(* CODESYS project stdnov.library
   Company: National Oilwell Varco
   DefaultNamespace: stdNOV
   Version: 1.0.0.2936
   Placeholder: stdNOV
   Author: AACD
   Title: stdNOV

Project tree, tasks and I/O mapping:
  libraries: SysTimeCore, * (System); Tc2_EtherCAT, * (Beckhoff Automation GmbH); Tc2_ModbusSrv, * (Beckhoff Automation GmbH); Tc2_Standard, * (Beckhoff Automation GmbH); Tc2_System, * (Beckhoff Automation GmbH); Tc2_Utilities, 3.3.41.0 (Beckhoff Automation GmbH); Util, * (System)
  10 Documentation/
  20 Program Organization Units/
    Alarms/
      function f_AlarmCode [ST]
      function f_DeviceId [ST]
      function f_FaultCode [ST]
      function f_GetFaultCodePriority [ST]
      function block fb_AlarmHandler [ST]: Clear, FB_exit, FB_init, GetAlarmCodeIndex, GetAlarms, GetNumOfActiveAlarms, GetNumOfAlarms, GetNumOfDeviceId, GetNumRegisteredCodes, GetRegisteredAlarmCodeDWORDListPointer, GetRegisteredAlarmCodeListPointer, GetRegisteredDeviceComponentIdListPointer, GetRegisteredDeviceElementIdListPointer, GetRegisteredFaultCondiitionIdListPointer, GetRegisteredFaultPriorityIdListPointer, Init, RegisterAlarmCode, Set
      function block fb_AlarmInterface [ST]: FB_exit, FB_init, ResetAlarms, UpdateAlarms
      function block fb_AlarmMonitor [ST]: CheckLimits, DisableLimit, EnableLimit, FB_exit, FB_init, GetState, InitAlarm, Monitor, MonitorBool, MonitorInt, MonitorReal, SetDelayOn, SetLimitBool, SetLimitInt, SetLimitReal
    Command Interface/
      Interfaces/
        interface i_commandHandler: CommandDone, CommandRunning, CommandStart, Fault, Reset
      function block fb_CommandInterface [ST]: CMD_ClearCommandBuffer, CMD_Fault, CMD_Init, CMD_IsCommandValid, CMD_Reset, CMD_SendCommand, CMD_SetTraceTable, CMD_TRACE, CMD_UpdateCommandInterface, ExecuteAction
    Control Functions/
      PID Functions/
        function block PID_StandAlone [ST]: Execute, FB_init, GetGains, GetLimits, init, Reset, SetGains, SetLimits
        function block PID_StandAlone_AntiWindup [ST]: Execute, FB_init, GetConfig, init, Reset, SetConfig
        function block PID_StandAlone_Stuck [ST]: Execute, FB_init, GetGains, GetLimits, init, Reset, SetGains, SetLimits
    Equipment Functions/
      TriStateValve/
        ENUMS/
          data type TriStateValveFsmAction
          data type TriStateValveFsmEvent
          data type TriStateValveFsmState
        function block fb_AnalogFeedbackValve [ST]: CloseValve, FB_exit, FB_init, InitAlarms, IsClosed, IsOpened, IsShifting, IsShiftingError, OpenValve
        function block fb_DigitalFeedbackDualActionValve [ST]: CloseValve, FB_exit, FB_init, InitAlarms, IsClosed, IsOpened, IsShifting, IsShiftingError, OpenValve
        function block fb_DigitalFeedbackSingleActionValve [ST]: CloseValve, FB_exit, FB_init, InitAlarms, IsClosed, IsOpened, IsShifting, IsShiftingError, OpenValve
        function block fb_DigitalFeedbackValve [ST]: CloseValve, FB_exit, FB_init, InitAlarms, IsClosed, IsOpened, IsShifting, IsShiftingError, OpenValve
        function block fb_NoFeedbackValve [ST]: CloseValve, FB_exit, FB_init, IsClosed, IsOpened, IsShifting, IsShiftingError, OpenValve
        function block fb_TriStateValve [ST]: CloseValve, ExecuteAction, FB_exit, FB_init, OpenValve
    FSM/
      Interfaces/
        interface i_actionHandler: ExecuteAction
      function block fb_FSM [ST]: FB_exit, FB_init, FSM_ASSERT, FSM_GetCurrentAction, FSM_GetCurrentEvent, FSM_GetCurrentState, FSM_GetNextState, FSM_GetPreviousState, FSM_ProcessEvent, FSM_ProcessEventWithParms, FSM_Reset, FSM_SetAlwaysChangeState, FSM_SetConditionalState, FSM_SetDebugTraceTable, FSM_SetErrorState, FSM_TRACE
    Input-Output Functions/
      function block fb_AnalogOutputActuator [ST]: AbortCal, Arm, Disarm, Fault, FB_exit, FB_init, GetDevId, GetMaxInput, GetMaxOutput, GetMinInput, GetMinOutput, GetZeroCalValue, InitAlarms, IsZeroCalRunning, ZeroCal
      function block fb_AnalogTransducer [ST]: AbortCal, Arm, Disarm, Fault, FB_exit, FB_init, GetDevId, GetMaxOutput, GetMinOutput, GetWireBreakStatus, GetZeroCalValue, InitAlarms, IsZeroCalRunning, ZeroCal
      function block fb_FreqTransducer [ST]: FaultHandlerSetOrClear, FB_init, GetDevId, InitAlarms
    Instrument-Controller Functions/
      function block fb_Densitometer [ST]: CalculateUserkFact, GetCorrectedDensitySGU, GetDensityRange_MinMax, GetRawDensity, GetUserKFact, InitAlarms, SetDensityRange_MinMax, SetRawDensity, setUserKFact
      function block fb_ENDP_Analog [ST]: FB_init, Get_UserAlarms, GetConfigData, GetRange_MinMax, InitAlarms, Scale, Set_Hysteresis, SetRange_MinMax, SetRange_UserAlarms
      function block fb_ENDP_AnalogCalPressure [ST]: CalculateUserKFactor, CalibrateHighDataPoint, CalibrateLowDataPoint, ClearCalibration, FB_Exit, FB_Init, GetConfigData, GetCorrectedPressure, GetLowerCalDataPoint, GetPressureRange, GetRawPressure, GetUpperCalDataPoint, GetUserAlarms, GetUserKFactor, InitAlarms, SetHysteresis, SetLowerCalDataPoint, SetPressureRange, SetRangeUserAlarms, SetRawPressure, SetUpperCalDataPoint, SetUserKFactor
      function block fb_ENDP_AnalogDensitometer [ST]: FB_exit, FB_init
      function block fb_ENDP_AnalogFlowmeter [ST]: CalibrateHighDataPoint, CalibrateLowDataPoint, ClearCalibration, FB_exit, FB_init, GetLowerCalDataPoint, GetUpperCalDataPoint, SetLowerCalDataPoint, SetUpperCalDataPoint
      function block fb_ENDP_Freq_Tachometer [ST]: FB_init
      function block fb_ENDP_FreqFlowmeter [ST]: FB_exit, FB_init, GetKFact, GetPPR, GetTimebase, SetKFact, SetPPR, SetTimebase
      function block fb_ENDP_SimulatedDensitometer [ST]: FB_exit, FB_init, SetSimDensity
      function block fb_ENDP_SimulatedFlowMeter [ST]: FB_exit, FB_init, SetSimFlow
      function block fb_FlowMeter [ST]: CalculateUserKFact, GetCorrectedFlow, GetFlowRange_MinMax, GetRawFlow, GetUserAlarms, GetUserKFact, GetVolumeTotal1, GetVolumeTotal2, GetVolumeTotal3, InitAlarms, PauseVolumeTotal1, PauseVolumeTotal2, PauseVolumeTotal3, ResetVolumeTotal1, ResetVolumeTotal2, ResetVolumeTotal3, ResumeVolumeTotal1, ResumeVolumeTotal2, ResumeVolumeTotal3, SetFlowRange_MinMax, SetRawFlow, SetUserAlarms, SetUserKFact
      function block fb_Indicator [ST]: FB_exit, FB_init, Off, On
      function block fb_STARTP_ControlActuator [ST]: FB_init, GetConfigData, GetRange_MinMax, Scale, Set_Hysteresis, SetRange_MinMax
      function block fb_Switch [ST]: Equals, FB_exit, FB_init, GetDebounce, SetDebounce
    Interlock Functions/
      function block fb_NOVInterlock [ST]: FB_exit, FB_init, InitAlarms
    Modbus/
      function block fb_ModbusError [FBD]
      function block fb_ModbusServer [FBD]: afterAccess, beforeAccess, FB_exit, FB_init, GetCoilPointer, GetDiscreteInputPointer, GetHoldingRegisterPointer, GetInputRegisterPointer, IsClientConnected, UpdateConnectionList
      function block fb_ReadHoldingRegisters [FBD]
      function block fb_ReadInputRegisters [FBD]
      function block fb_WriteHoldingRegisters [FBD]
    Process Calculation Functions/
      function f_CalculateDensityPPAfromSGU [ST]
      function f_CalculateDensityPPGfromSGU [ST]
    Testing Functions/
      function block FB_CNTRLSYS_RESPONSE [ST]
      function block fb_TriStateValveSimulator [ST]
    Utility Functions/
      Conversion Functions/
        function F_SPLIT_REGISTERS [ST]
        function F_STATUS_WORD_TO_WORD [ST]
      Statistic Functions/
        function block FB_RUNNING_AVG [ST]
      function f_LinearScale [ST]
      function block fb_Clock [ST]
      function block fb_ElapsedTime [ST]: FB_exit, FB_init, GetElapsedLTime, GetElapsedTime, StartNow
      function block fb_ElapseTimer [ST]: FB_exit, FB_init, Freeze, Initialize, Reset
      function block fb_FilterExp [ST]: FB_exit, FB_init, GetSampleSize, Initialize, SetSampleSize
      function block fb_GetCycleTime [ST]
      function block fb_TriggerTimer [ST]
      function block Logger [ST]: getCount, LogPoint
      function block Totalizer [ST]: Disable, Enable, FB_Init, Reset, SetTotal
  40 Data Types/
    Alarm Interface Types/
      data type TAlarm
      data type TAlarmData
    Alarm Types/
      global variables GLOBAL_ALARMS
      data type TAlarmCode
      data type TAlarmLimit
      data type TAlarmMessage
      data type TAlarmMonitorType
      data type TAlarmType
      data type TComponentId
      data type TDeviceId
      data type TElementId
      data type TFaultCode
      data type TFaultCondition
      data type TFaultPriority
      data type UAlarmCode
      data type UDeviceId
      data type UFaultCode
    Command Interface/
      data type Command_FsmAction
      data type Command_FsmDebugTableEntry
      data type Command_FsmEvent
      data type Command_FsmState
      data type TControlCommand
      data type TControlCommandBuffer
      data type TControlCommandParms
      data type TControlCommandResponse
      data type TControlResponse
      data type TControlResponseMessage
    Equipment Types/
      data type TValveShutoff
      data type TValveTriStatePosition
    FSM Types/
      global variables GLOBAL_FSM
      data type TFsmAction
      data type TFsmDebugTableEntry
      data type TFsmError
      data type TFsmEvent
      data type TFsmEventDesc
      data type TFsmEventQIndex
      data type TFsmState
    Generic Types/
      data type ST_Bits
    Input-Output Types/
      data type AI_ChannelInputs
      data type AO_ChannelOutputs
      data type Freq_ChannelInput
    Instrument-Controller Types/
      global variables GLOBAL_INSTRUMENTS
      data type HmiGaugeState
      data type TCalibrationDataPoint
      data type TEndPoint
      data type TEndPointConfig
      data type TEnuHmiGaugeState
    Interlock Types/
      data type THMINOVInterlock
      data type TNOVInterlockCmdBypassInWORD
      data type TNOVInterlockIn
      data type TNOVInterlockStatusInWORD
      data type TNOVInterlockStatusOut
      data type TNOVInterlockStatusOutWORD
    Modbus Types/
      global variables GLOBAL_MODBUS
      data type TModbusServerConfig
      data type TModbusServerConnection
      data type TModbusTargetConfig
    Utility Types/
      data type DataPoint
      data type TGenericStatusWord
    global variables GLOBAL_CONSTANTS
  80 Status/
  Project Information/
    function F_GetCompany [ST]
    function F_GetTitle [ST]
    function F_GetVersion [ST]
  Version/
    global variables Global_Version
*)

// 20 Program Organization Units/Equipment Functions/TriStateValve/ENUMS/TriStateValveFsmAction
{attribute 'qualified_only'}
//{attribute 'strict'}
TYPE TriStateValveFsmAction :
(
	FsmAction_None := FSM_ACTION_NONE,		(*0*)
	FsmAction_ValveEnabled := 1,			(*1*)
	FsmAction_ValveDisabled,				(*2*)
	FsmAction_ValveOpen,					(*3*)
	FsmAction_ValveClose,					(*4*)
	FsmAction_ValveOpened,					(*5*)
	FsmAction_ValveClosed,					(*6*)
	FsmAction_ValveShiftTimerExpired,		(*7*)
	FsmAction_ValvePositionMismatch,		(*8*)
	NUM_FsmTriStateValveActions				(*9*)
) BYTE;
END_TYPE

// 20 Program Organization Units/Equipment Functions/TriStateValve/ENUMS/TriStateValveFsmEvent
{attribute 'qualified_only'}
//{attribute 'strict'}
TYPE TriStateValveFsmEvent :
(
	FsmEvent_ValveEnable := 0,			(*0*)
	FsmEvent_ValveDisable,				(*1*)
	FsmEvent_ValveOpen,					(*2*)
	FsmEvent_ValveClose,				(*3*)
	FsmEvent_ValveOpened,				(*4*)
	FsmEvent_ValveClosed,				(*5*)
	FsmEvent_ValveShiftTimerExpired,	(*6*)
	FsmEvent_ValvePositionMismatch,		(*7*)
	NUM_FsmTriStateValveEvents			(*8*)
) BYTE;
END_TYPE

// 20 Program Organization Units/Equipment Functions/TriStateValve/ENUMS/TriStateValveFsmState
{attribute 'qualified_only'}
//{attribute 'strict'}
TYPE TriStateValveFsmState :
(
	FsmState_Error := 0,			(*0*)
	FsmState_ValveOff,				(*1*)
	FsmState_ValveClosed,			(*2*)
	FsmState_ValveOpened,  			(*3*)
	FsmState_ValveShifting,			(*4*)
	NUM_FsmTriStateValveStates		(*5*)
) BYTE;
END_TYPE

// 40 Data Types/Alarm Interface Types/TAlarm
TYPE TAlarm :
STRUCT
	code	: UDINT;
	state	: BOOL;
	ack		: BOOL;
	message	: STRING(95);
END_STRUCT
END_TYPE

// 40 Data Types/Alarm Interface Types/TAlarmData
TYPE TAlarmData :
STRUCT
	NumOfAlarms			: INT;
	NumOfActiveAlarms	: INT;
	RefreshAlarms		: BOOL;
	AlarmState			: INT;
	Alarm				: ARRAY[0.._ALARM_ARRAY_MAX_SIZE] OF TAlarm;
END_STRUCT
END_TYPE

// 40 Data Types/Alarm Types/TAlarmCode
// I have made the DeviceId the MSB so that when sorting the alarm list
// all similar deviceId's will be grouped together. <JAISON>
TYPE TAlarmCode :
STRUCT
	faultCode	: UFaultCode;	// LSB (16 bits)
	devId		: UDeviceId;	// MSB (16 bits)
END_STRUCT
END_TYPE

// 40 Data Types/Alarm Types/TAlarmLimit
TYPE TAlarmLimit :
STRUCT
	limitOn		: LREAL;
	limitOff	: LREAL;
	enable		: BOOL;
	monitorType	: TAlarmMonitorType;
END_STRUCT
END_TYPE

// 40 Data Types/Alarm Types/TAlarmMessage
TYPE TAlarmMessage :
STRUCT
	code	: UAlarmCode;			// 32 bits
	msg		: STRING;
END_STRUCT
END_TYPE

// 40 Data Types/Alarm Types/TAlarmMonitorType
{attribute 'qualified_only'}
{attribute 'strict'}
TYPE TAlarmMonitorType :
(
	lower_limit := 0,
	upper_limit
);
END_TYPE

// 40 Data Types/Alarm Types/TAlarmType
TYPE TAlarmType :
STRUCT
	code	: UAlarmCode;
	state	: BOOL;
	message	: STRING;
END_STRUCT
END_TYPE

// 40 Data Types/Alarm Types/TComponentId
TYPE TComponentId : BYTE; END_TYPE

// 40 Data Types/Alarm Types/TDeviceId
// Device Ids (16 bits)
TYPE TDeviceId :
STRUCT
	element		: BYTE;	// LSB (8 bits)
	component	: BYTE;	// MSB (8 bits)
END_STRUCT
END_TYPE

// 40 Data Types/Alarm Types/TElementId
TYPE TElementId : BYTE; END_TYPE

// 40 Data Types/Alarm Types/TFaultCode
// Fault Codes (16 bits)
TYPE TFaultCode :
STRUCT
	condition	: BYTE; // LSB (8 bits)
	priority	: BYTE; // MSB (8 bits) 	
END_STRUCT
END_TYPE

// 40 Data Types/Alarm Types/TFaultCondition
{attribute 'qualified_only'}
//{attribute 'strict'}
TYPE TFaultCondition :
(
	SelfTest := 0,
	Generic,
	Check,
	Config,
	UnderLimit,
	OverLimit,
	Protect,
	UnderWarning,
	OverWarning,
	TimeOut,
	HwError,
	ShortCircuit,
	UnderRange,
	OverRange,
	Shutdown,
	Stop,
	Interlock
) BYTE;
END_TYPE

// 40 Data Types/Alarm Types/TFaultPriority
{attribute 'qualified_only'}
//{attribute 'strict'}
TYPE TFaultPriority :
(
	// The 2 most significant bits of the fault code are reserved for severity
	// This has now been explanded to 8 bits however the Hex values are kept for
	// backwards compatibility AND to give space for future priority additions. <JAISON>
	Information := 16#00,	// 0
	Warning		:= 16#40,	// 64
	Error		:= 16#80,	// 128
	Reserved	:= 16#C0,	// 192
	Critical	:= 16#FF	// 255
) BYTE;
END_TYPE

// 40 Data Types/Alarm Types/UAlarmCode
TYPE UAlarmCode :
UNION
	code		: TAlarmCode;
	code_UDINT	: UDINT;
	code_DWORD	: DWORD;
	code_BYTES	: ARRAY[1..4] OF BYTE;   
    code_BITS	: ARRAY[1..4] OF ST_Bits;
END_UNION
END_TYPE

// 40 Data Types/Alarm Types/UDeviceId
TYPE UDeviceId :
UNION
	devId		: TDeviceId;
	devId_UINT	: UINT;
	devId_WORD	: WORD;
	devId_BYTES	: ARRAY[1..2] OF BYTE;  
    devId_BITS	: ARRAY[1..2] OF ST_Bits;
END_UNION
END_TYPE

// 40 Data Types/Alarm Types/UFaultCode
TYPE UFaultCode :
UNION
	faultcode		: TFaultCode;
	faultcode_UINT	: UINT;
	faultcode_WORD	: WORD;
	faultcode_BYTES	: ARRAY[1..2] OF BYTE;   
    faultcode_BITS	: ARRAY[1..2] OF ST_Bits;
END_UNION
END_TYPE

// 40 Data Types/Command Interface/Command_FsmAction
{attribute 'qualified_only'}
//{attribute 'strict'}
TYPE Command_FsmAction :
(
	FsmAction_None := FSM_ACTION_NONE,				(*0*)
	FsmAction_EnableControl := 1,					(*1*)
	FsmAction_DisableControl,						(*2*)
	FsmAction_RunCommand,							(*3*)
	FsmAction_CommandDone,							(*4*)
	FsmAction_Fault,								(*5*)
	FsmAction_Reset,								(*6*)
	NUM_FsmCommandInterfaceActions					(*7*)
) BYTE;
END_TYPE

// 40 Data Types/Command Interface/Command_FsmDebugTableEntry
TYPE Command_FsmDebugTableEntry :
STRUCT
	state		: Command_FsmState;	// State transitioning to
	event		: Command_FsmEvent;	// Event causing the transition
	timeInState	: UDINT;			// Elapsed time since the last event (ms)
END_STRUCT
END_TYPE

// 40 Data Types/Command Interface/Command_FsmEvent
{attribute 'qualified_only'}
//{attribute 'strict'}
TYPE Command_FsmEvent :
(
	FsmEvent_ControlEnable := 0,		(*0*)
	FsmEvent_ControlDisable,			(*1*)
	FsmEvent_RunCommand,				(*2*)
	FsmEvent_CommandDone,				(*3*)
	FsmEvent_Fault,						(*4*)
	FsmEvent_Reset,						(*5*)
	NUM_FsmCommandInterfaceEvents		(*6*)
) BYTE;
END_TYPE

// 40 Data Types/Command Interface/Command_FsmState
{attribute 'qualified_only'}
//{attribute 'strict'}
TYPE Command_FsmState :
(
	FsmState_ControlFault := 0,			(*0*)
	FsmState_ControlDisabled,			(*1*)
	FsmState_CommandRunning,			(*2*)
	FsmState_ControlReady,				(*3*)
	NUM_FsmCommandInterfaceStates		(*4*)	
) BYTE;
END_TYPE

// 40 Data Types/Command Interface/TControlCommand
{attribute 'strict'}
TYPE TControlCommand : INT; END_TYPE

// 40 Data Types/Command Interface/TControlCommandBuffer
TYPE TControlCommandBuffer :
STRUCT
	command		: TControlCommand;
	parms		: TControlCommandParms;
	response	: TControlCommandResponse;
END_STRUCT
END_TYPE

// 40 Data Types/Command Interface/TControlCommandParms
TYPE TControlCommandParms : ARRAY[1..12] OF WORD; END_TYPE

// 40 Data Types/Command Interface/TControlCommandResponse
TYPE TControlCommandResponse :
STRUCT
	response	: TControlResponse;
	message		: TControlResponseMessage;
END_STRUCT
END_TYPE

// 40 Data Types/Command Interface/TControlResponse
{attribute 'strict'}
TYPE TControlResponse : INT; END_TYPE

// 40 Data Types/Command Interface/TControlResponseMessage
TYPE TControlResponseMessage : STRING(27); END_TYPE

// 40 Data Types/Equipment Types/TValveShutoff
TYPE TValveShutoff :
STRUCT
	Open	: BOOL;
	Close	: BOOL;
END_STRUCT
END_TYPE

// 40 Data Types/Equipment Types/TValveTriStatePosition
{attribute 'qualified_only'}
{attribute 'strict'}
TYPE TValveTriStatePosition :
(
	PosClosed := 0,
	PosOpened,
	PosUnknown
);
END_TYPE

// 40 Data Types/FSM Types/TFsmAction
TYPE TFsmAction : BYTE; END_TYPE

// 40 Data Types/FSM Types/TFsmDebugTableEntry
TYPE TFsmDebugTableEntry :
STRUCT
	state		: TFsmState;	// State transitioning to
	event		: TFsmEvent;	// Event causing the transition
	timeInState	: UDINT;		// Elapsed time since the last event (ms)
END_STRUCT
END_TYPE

// 40 Data Types/FSM Types/TFsmError
{attribute 'qualified_only'}
TYPE TFsmError :
(
	FSM_ERROR_NONE := 0,
	FSM_INVALID_NEXT_STATE,
	FSM_PARM_SIZE_ERROR,
	FSM_EVENT_Q_SIZE_ERROR,
	FSM_INVALID_EVENT_ERROR,
	FSM_INVALID_ACTION,
	FSM_INVALID_CONDITIONAL_STATE,
	FSM_INVALID_ERROR_STATE
) BYTE;
END_TYPE

// 40 Data Types/FSM Types/TFsmEvent
{attribute 'strict'}
TYPE TFsmEvent : BYTE; END_TYPE

// 40 Data Types/FSM Types/TFsmEventDesc
TYPE TFsmEventDesc :
STRUCT
	event		: BYTE;
	parms		: POINTER TO BYTE;
	parmSize	: UINT;
END_STRUCT
END_TYPE

// 40 Data Types/FSM Types/TFsmEventQIndex
TYPE TFsmEventQIndex : UINT; END_TYPE

// 40 Data Types/FSM Types/TFsmState
TYPE TFsmState : BYTE; END_TYPE

// 40 Data Types/Generic Types/ST_Bits
TYPE ST_Bits :
STRUCT
	bBit1  : BIT;
    bBit2  : BIT;
    bBit3  : BIT;
    bBit4  : BIT;
    bBit5  : BIT;
    bBit6  : BIT;
    bBit7  : BIT;
    bBit8  : BIT;   
END_STRUCT
END_TYPE

// 40 Data Types/Input-Output Types/AI_ChannelInputs
TYPE AI_ChannelInputs :
STRUCT
	value				: INT;
	underRange			: BOOL;
	overRange			: BOOL;
	error				: BOOL;
	shortCircuit		: BOOL;
END_STRUCT
END_TYPE

// 40 Data Types/Input-Output Types/AO_ChannelOutputs
TYPE AO_ChannelOutputs :
STRUCT
	value				: INT;
END_STRUCT
END_TYPE

// 40 Data Types/Input-Output Types/Freq_ChannelInput
TYPE Freq_ChannelInput :
STRUCT
	value		: DINT;
	//error		: BOOL;
END_STRUCT
END_TYPE

// 40 Data Types/Instrument-Controller Types/HmiGaugeState
{attribute 'qualified_only'}
{attribute 'strict'}
TYPE HmiGaugeState :
(
	LowAlarm := -2,
	LowWarning := -1,
	No_Alarm := 0,
	HighWarning := 1,
	HighAlarm := 2
);
END_TYPE

// 40 Data Types/Instrument-Controller Types/TCalibrationDataPoint
TYPE TCalibrationDataPoint :
STRUCT
	yValue	: REAL;
	xValue	: REAL;
END_STRUCT
END_TYPE

// 40 Data Types/Instrument-Controller Types/TEndPoint
TYPE TEndPoint :
STRUCT
	Value	:	REAL;
	State	:	INT;
END_STRUCT
END_TYPE

// 40 Data Types/Instrument-Controller Types/TEndPointConfig
TYPE TEndPointConfig :
STRUCT
	MinValue	:	REAL;
	MaxValue	:	REAL;
	OffsetValue	:	REAL;
	LowLimit	:	REAL;
	HighLimit	:	REAL;
	LowWarning	:	REAL;
	HighWarning	:	REAL;
END_STRUCT
END_TYPE

// 40 Data Types/Instrument-Controller Types/TEnuHmiGaugeState
{attribute 'qualified_only'}
{attribute 'strict'}
TYPE TEnuHmiGaugeState :
(
	LowAlarm 	:= -2,
	LowWarning 	:= -1,
	No_Alarm 	:= 0,
	HighWarning	:= 1,
	HighAlarm 	:= 2
);
END_TYPE

// 40 Data Types/Interlock Types/THMINOVInterlock
/// WORD ALLIGNED (2 WORDS) <GRAHAM>
TYPE THMINOVInterlock :
STRUCT
	
	//HMIInterlockBypass : TNOVInterlockCmdBypassInWORD;	// INTLK DynIn, for future use, HMI may have the ability to override in the future
	HMIInterlockProcessed: TNOVInterlockStatusOutWORD; 		// INTLK DynOut
	
END_STRUCT
END_TYPE

// 40 Data Types/Interlock Types/TNOVInterlockCmdBypassInWORD
/// this input commmand data structure word is for future use (not used currently) <GRAHAM>
TYPE TNOVInterlockCmdBypassInWORD :
STRUCT
	
	IntlkBypassALL	: BIT; // Bypass/override all interlocks command input
	Intlk01Bypass	: BIT; // TRUE = (OVERRIDE ACTIVE), FALSE = (OVERRIDE NOT ACTIVE)
	Intlk02Bypass	: BIT; // TRUE = (OVERRIDE ACTIVE), FALSE = (OVERRIDE NOT ACTIVE)
	Intlk03Bypass	: BIT; // TRUE = (OVERRIDE ACTIVE), FALSE = (OVERRIDE NOT ACTIVE)
	Intlk04Bypass	: BIT; // TRUE = (OVERRIDE ACTIVE), FALSE = (OVERRIDE NOT ACTIVE)
	Intlk05Bypass	: BIT; // TRUE = (OVERRIDE ACTIVE), FALSE = (OVERRIDE NOT ACTIVE)
	Intlk06Bypass	: BIT; // TRUE = (OVERRIDE ACTIVE), FALSE = (OVERRIDE NOT ACTIVE)
	Intlk07Bypass	: BIT; // TRUE = (OVERRIDE ACTIVE), FALSE = (OVERRIDE NOT ACTIVE)
	Intlk08Bypass	: BIT; // TRUE = (OVERRIDE ACTIVE), FALSE = (OVERRIDE NOT ACTIVE)
	Intlk09Bypass	: BIT; // TRUE = (OVERRIDE ACTIVE), FALSE = (OVERRIDE NOT ACTIVE)
	Intlk10Bypass	: BIT; // TRUE = (OVERRIDE ACTIVE), FALSE = (OVERRIDE NOT ACTIVE)
	Intlk11Bypass	: BIT; // TRUE = (OVERRIDE ACTIVE), FALSE = (OVERRIDE NOT ACTIVE)
	Intlk12Bypass	: BIT; // TRUE = (OVERRIDE ACTIVE), FALSE = (OVERRIDE NOT ACTIVE)
	Intlk13Bypass	: BIT; // TRUE = (OVERRIDE ACTIVE), FALSE = (OVERRIDE NOT ACTIVE)
	IntlkBypassNONE	: BIT; // Do not Bypass/override any interlocks command input
	Bit15			: BIT; // Spare Bit command input
END_STRUCT
END_TYPE

// 40 Data Types/Interlock Types/TNOVInterlockIn
/// WORD ALLIGNED (2 WORDS), this input data structure is for future use (not used currently) <GRAHAM>
TYPE TNOVInterlockIn :
STRUCT
	
	InterlockStatus		: TNOVInterlockStatusInWORD;	// INTLK In (from NOV or NSA interlocks)
	//InterlockBypass	: TNOVInterlockCmdBypassInWORD;	// INTLK In (from an external device), for future use
	
END_STRUCT
END_TYPE

// 40 Data Types/Interlock Types/TNOVInterlockStatusInWORD
/// this input structure data word is for future use (not used currently) <GRAHAM>
TYPE TNOVInterlockStatusInWORD :
STRUCT
	
	Bit0	: BIT; // Not Defined
	Intlk01	: BIT; // TRUE = (INTLK SATISFIED), FALSE = (INTLK NOT SATISFIED)
	Intlk02	: BIT; // TRUE = (INTLK SATISFIED), FALSE = (INTLK NOT SATISFIED)
	Intlk03	: BIT; // TRUE = (INTLK SATISFIED), FALSE = (INTLK NOT SATISFIED)
	Intlk04	: BIT; // TRUE = (INTLK SATISFIED), FALSE = (INTLK NOT SATISFIED) 
	Intlk05	: BIT; // TRUE = (INTLK SATISFIED), FALSE = (INTLK NOT SATISFIED)
	Intlk06	: BIT; // TRUE = (INTLK SATISFIED), FALSE = (INTLK NOT SATISFIED)
	Intlk07	: BIT; // TRUE = (INTLK SATISFIED), FALSE = (INTLK NOT SATISFIED)
	Intlk08	: BIT; // TRUE = (INTLK SATISFIED), FALSE = (INTLK NOT SATISFIED)
	Intlk09	: BIT; // TRUE = (INTLK SATISFIED), FALSE = (INTLK NOT SATISFIED)
	Intlk10	: BIT; // TRUE = (INTLK SATISFIED), FALSE = (INTLK NOT SATISFIED)
	Intlk11	: BIT; // TRUE = (INTLK SATISFIED), FALSE = (INTLK NOT SATISFIED)
	Intlk12	: BIT; // TRUE = (INTLK SATISFIED), FALSE = (INTLK NOT SATISFIED)
	Intlk13	: BIT; // TRUE = (INTLK SATISFIED), FALSE = (INTLK NOT SATISFIED)
	Bit14	: BIT; // Not defined
	Bit15	: BIT; // Not defined
	
END_STRUCT
END_TYPE

// 40 Data Types/Interlock Types/TNOVInterlockStatusOut
/// WORD ALLIGNED (1 WORD), // this seperate output structure data word is for future use (not used currently) <GRAHAM>
TYPE TNOVInterlockStatusOut :
STRUCT
	
	InterlockProcessed: TNOVInterlockStatusOutWORD; // INTLK DynOut
END_STRUCT
END_TYPE

// 40 Data Types/Interlock Types/TNOVInterlockStatusOutWORD
TYPE TNOVInterlockStatusOutWORD :
STRUCT
	IntlkOK_NoBypass	: BIT; 	// All interlocks are Ok with no bypasses/overrides
	Intlk01				: BIT; // TRUE = (INTLK IS TRUE OR OVERRIDE IS TRUE IF OVERRIDE IS ACTIVE, FALSE = (INTLK IS FALSE AND OVERRIDE IS FALSE IF OVERRIDE IS ACTIVE)
	Intlk02				: BIT; // TRUE = (INTLK IS TRUE OR OVERRIDE IS TRUE IF OVERRIDE IS ACTIVE, FALSE = (INTLK IS FALSE AND OVERRIDE IS FALSE IF OVERRIDE IS ACTIVE)
	Intlk03				: BIT; // TRUE = (INTLK IS TRUE OR OVERRIDE IS TRUE IF OVERRIDE IS ACTIVE, FALSE = (INTLK IS FALSE AND OVERRIDE IS FALSE IF OVERRIDE IS ACTIVE)
	Intlk04				: BIT; // TRUE = (INTLK IS TRUE OR OVERRIDE IS TRUE IF OVERRIDE IS ACTIVE, FALSE = (INTLK IS FALSE AND OVERRIDE IS FALSE IF OVERRIDE IS ACTIVE)
	Intlk05				: BIT; // TRUE = (INTLK IS TRUE OR OVERRIDE IS TRUE IF OVERRIDE IS ACTIVE, FALSE = (INTLK IS FALSE AND OVERRIDE IS FALSE IF OVERRIDE IS ACTIVE)
	Intlk06				: BIT; // TRUE = (INTLK IS TRUE OR OVERRIDE IS TRUE IF OVERRIDE IS ACTIVE, FALSE = (INTLK IS FALSE AND OVERRIDE IS FALSE IF OVERRIDE IS ACTIVE)
	Intlk07				: BIT; // TRUE = (INTLK IS TRUE OR OVERRIDE IS TRUE IF OVERRIDE IS ACTIVE, FALSE = (INTLK IS FALSE AND OVERRIDE IS FALSE IF OVERRIDE IS ACTIVE)
	Intlk08				: BIT; // TRUE = (INTLK IS TRUE OR OVERRIDE IS TRUE IF OVERRIDE IS ACTIVE, FALSE = (INTLK IS FALSE AND OVERRIDE IS FALSE IF OVERRIDE IS ACTIVE)
	Intlk09				: BIT; // TRUE = (INTLK IS TRUE OR OVERRIDE IS TRUE IF OVERRIDE IS ACTIVE, FALSE = (INTLK IS FALSE AND OVERRIDE IS FALSE IF OVERRIDE IS ACTIVE)
	Intlk10				: BIT; // TRUE = (INTLK IS TRUE OR OVERRIDE IS TRUE IF OVERRIDE IS ACTIVE, FALSE = (INTLK IS FALSE AND OVERRIDE IS FALSE IF OVERRIDE IS ACTIVE)
	Intlk11				: BIT; // TRUE = (INTLK IS TRUE OR OVERRIDE IS TRUE IF OVERRIDE IS ACTIVE, FALSE = (INTLK IS FALSE AND OVERRIDE IS FALSE IF OVERRIDE IS ACTIVE)
	Intlk12				: BIT; // TRUE = (INTLK IS TRUE OR OVERRIDE IS TRUE IF OVERRIDE IS ACTIVE, FALSE = (INTLK IS FALSE AND OVERRIDE IS FALSE IF OVERRIDE IS ACTIVE)
	Intlk13				: BIT; // TRUE = (INTLK IS TRUE OR OVERRIDE IS TRUE IF OVERRIDE IS ACTIVE, FALSE = (INTLK IS FALSE AND OVERRIDE IS FALSE IF OVERRIDE IS ACTIVE)
	IntlkOK_WithBypass	: BIT; // All interlocks are Ok with bypasses/overrides
	Bit15				: BIT; // Not defined
END_STRUCT
END_TYPE

// 40 Data Types/Modbus Types/TModbusServerConfig
TYPE TModbusServerConfig :
STRUCT
	xInstalled				: BOOL;
	tTimeOut				: TIME;
END_STRUCT
END_TYPE

// 40 Data Types/Modbus Types/TModbusServerConnection
TYPE TModbusServerConnection :
STRUCT
	xActive					: BOOL;
	ipAddress				: STRING(20);
	bUnitId					: BYTE;		
	bFunctionCode			: BYTE;
	wReadAddress			: WORD;
	uiReadQuantity			: UINT;
	uiReadQuantityTotal		: UINT;
	wWriteAddress			: WORD;
	uiWriteQuantity			: UINT;
	uiWriteQuantityTotal	: UINT;
	commLossTimer			: TON;
END_STRUCT
END_TYPE

// 40 Data Types/Modbus Types/TModbusTargetConfig
TYPE TModbusTargetConfig :
STRUCT
	xInstalled				: BOOL;			// Not Used
	sIPAddr					: STRING(23);
	wTCPPort				: WORD;
	bUnitID					: BYTE;
	tTimeOut				: TIME;
END_STRUCT
END_TYPE

// 40 Data Types/Utility Types/DataPoint
TYPE DataPoint :
STRUCT
	timestamp: TIME;
	message: STRING(20);
	counter: UINT;
END_STRUCT
END_TYPE

// 40 Data Types/Utility Types/TGenericStatusWord
/// Generic Status Word to handle Word to Bit
TYPE TGenericStatusWord :
STRUCT
	bit0: BIT;
	bit1: BIT;
	bit2: BIT;
	bit3: BIT;
	bit4: BIT;
	bit5: BIT;
	bit6: BIT;
	bit7: BIT;
	bit8: BIT;
	bit9: BIT;
	bit10: BIT;
	bit11: BIT;
	bit12: BIT;
	bit13: BIT;
	bit14: BIT;
	bit15: BIT;
END_STRUCT
END_TYPE

// 40 Data Types/Alarm Types/GLOBAL_ALARMS
{attribute 'global_init_slot' := '49987'}
VAR_GLOBAL CONSTANT
	
	(* --------------------------------------------------------------------------
	Config Parm : _ALARM_ARRAY_MAX_SIZE
	Description : 	This option defines the maximum number of elements defined in 
				 	all of the defined alarm arrays.  This includes the following:
						fb_AlarmHandler/m_alarmList - Internal alarm list
						fb_AlarmInterface/FB_Init/alarmMsg - Static Alarm message array
						fb_AlarmInterface/UpdateAlarms/m_pAlarms - Alarm Interface array
	Notes       : 	This value should be set greater than the maximum number of
					defined alarms in the system.
	-------------------------------------------------------------------------- *)
	_ALARM_ARRAY_MAX_SIZE: UINT := 400;
	
END_VAR

VAR_GLOBAL
	
	// Singleton Alarm handler instantiation
	// Use a pointer to this function block to access its methods
	gAlarmHandler		: fb_AlarmHandler;

END_VAR

// 40 Data Types/FSM Types/GLOBAL_FSM
{attribute 'global_init_slot' := '49987'}
VAR_GLOBAL CONSTANT
	
	(* --------------------------------------------------------------------------
	Config Parm : _FSM_EVENT_Q_SIZE
	Description : This option defines the number of events that can be
   		          stored by the Fsm.
	Notes       : This should be set to the largest queue size for all 
            	  FSMs in the system if optimization is required.
	              Maximum queue size is 256.
	-------------------------------------------------------------------------- *)
	_FSM_EVENT_Q_SIZE: UINT := 32;
	
	(* ---------------------------------------------------------------------------
	Config Parm : _FSM_MAX_PARM_STRUCT_SIZE
	Description : This option defines the maximum number of bytes required
            	  to store event parmeters.      
	Notes       : The size defaults to a large value to allow all event 
            	  parameters to be handled. This should be set to the largest
            	  parameter size for all events for all FSMs in the system if
           	   optimization is required.
	--------------------------------------------------------------------------- *)
	_FSM_MAX_PARM_STRUCT_SIZE: UINT := 512;
	
	(* --------------------------------------------------------------------------
	Config Parm : _FSM_ALLOW_CONDITIONAL_STATES
	Description : This option enables the handling of conditional states.
	Notes       : A conditional state is a state that has state transitions
 	             that can occur from within an action handler.
	-------------------------------------------------------------------------- *)
	_FSM_ALLOW_CONDITIONAL_STATES: BOOL := TRUE;
						
	(* ----------------------------------------------------------------------------
	Const name  : FSM_STATE_CONDITIONAL
	Description : Signifies that the next state is set by an action function 
	Notes       : Used in FSM table definitions
	---------------------------------------------------------------------------- *)
	FSM_STATE_CONDITIONAL: BYTE := 16#7F;

	(* ----------------------------------------------------------------------------
	Const name  : FSM_STATE_INVALID
	Description : Denotes that the state value is invalid
	Notes       : Returned by FSM_GetCurrentState()
	---------------------------------------------------------------------------- *)
	FSM_STATE_INVALID: BYTE := 16#FF;

	(* ----------------------------------------------------------------------------
	Const name  : FSM_EVENT_INVALID
	Description : Signifies that the event is not handled in the state 
	Notes       : Used in FSM table definitions
	---------------------------------------------------------------------------- *)
	FSM_EVENT_INVALID: BYTE := 16#FF;

	(* ----------------------------------------------------------------------------
	Const name  : FSM_ACTION_NONE
	Description : Signifies that no action is required to run
	              in the processing of the current state.
	Notes       : Used in FSM table definitions. For single action tables,
	              informs the FSM to move to the outlined next state.
	---------------------------------------------------------------------------- *)
	FSM_ACTION_NONE: BYTE := 16#00;
	
	(* ----------------------------------------------------------------------------
	Const name  : FSM_ACTION_UNEXPECTED_EVENT
	Description : Signifies that the event is not expected in the state 
	Notes       : Used in FSM table definitions and action handler. 
				  The FSM will not change state when this action is found.
	---------------------------------------------------------------------------- *)
	FSM_ACTION_UNEXPECTED_EVENT: BYTE := 16#FE;
	
	(* ----------------------------------------------------------------------------
	Const name  : FSM_ACTION_ERROR_EVENT
	Description : Signifies that an FSM Assert has failed 
	Notes       : Used in FSM action handler to trap actions required to run
				  on transition to the defined error state.  This will NOT be
				  called if no error state is defined.
	---------------------------------------------------------------------------- *)
	FSM_ACTION_ERROR_EVENT: BYTE := 16#FF;
	
END_VAR

// 40 Data Types/Instrument-Controller Types/GLOBAL_INSTRUMENTS
{attribute 'global_init_slot' := '49987'}
VAR_GLOBAL CONSTANT
	(* --------------------------------------------------------------------------
	Config Parm : NOTUSED
	Description : a flag-type-of-Value passed to ENDPoints to mark that
	              parameter is a Non-Value, rather a flag that is is unused.
				  It is definitely out of range foreseable usable-values,
				  and in addition it has a fraction part to eliminate coincidence.
	Notes       : This removes potential confusion with setting alarmable-limits 
            	  with a barrage of large values like a 100000.0 ...
                  or negatives if parameter is marking a LowAlarm side.
                  Felipe did that as a !quick! solution to place unreachable values
                  and thus mark them as "unused", but later it raised a LOT of questions
                  when we were standardizing that bckhff-code into Codesys as a library
	-------------------------------------------------------------------------- *)
	NOTUSED : REAL := 200001.24681;
	NOTUSED_HIMAX : REAL := (1000000.0);
	NOTUSED_LOMAX : REAL := (-300.0);
	
END_VAR

// 40 Data Types/Modbus Types/GLOBAL_MODBUS
{attribute 'global_init_slot' := '49987'}
VAR_GLOBAL CONSTANT
	
	// Static arrays can have a defined size from 0 - 65535.
	// The array index determines the modbus address for accessing the data. <JAISON>
	// I have left the "Discrete Input" and "Coil" array sizes smaller as its less likely we will use them
	// so no reason to waste memory space. <JAISON>
	DISCRETE_INPUT_ARRAY_SIZE		: UINT := 1;
	COIL_ARRAY_SIZE					: UINT := 1;
	INPUT_REGISTERS_ARRAY_SIZE		: UINT := 65535;
	HOLDING_REGISTERS_ARRAY_SIZE	: UINT := 65535;
	
END_VAR

VAR_GLOBAL
	
	// As long as the PLC Modbus server has been configured with the standard XML these arrays will be mapped to the server.
	// These memory spaces are to be accessed via the pointer using the "Get" routines of the fb_ModbusServer. <JAISON>
	gaxDiscreteInputs				: ARRAY [0..DISCRETE_INPUT_ARRAY_SIZE] OF BOOL;		// Internal modbus server discrete inputs memory space
	gaxCoils						: ARRAY [0..COIL_ARRAY_SIZE] OF BOOL;				// Internal modbus server coils memory space
	gawInputRegisters				: ARRAY [0..INPUT_REGISTERS_ARRAY_SIZE] OF WORD;	// Internal modbus server input register memory space
	gawHoldingRegisters				: ARRAY [0..HOLDING_REGISTERS_ARRAY_SIZE] OF WORD;	// Internal modbus server holding register memory space
	

END_VAR

// 40 Data Types/GLOBAL_CONSTANTS
{attribute 'global_init_slot' := '49987'}
VAR_GLOBAL CONSTANT

	(* --------------------------------------------------------------------------
	Constant	 : _NULL
	Description : This defines a common variable to test for NULL pointers.
	Notes       : 
	-------------------------------------------------------------------------- *)
	_NULL: UINT := 0;
	
	(* C O N V E R S I O N   F A C T O R S *)
	PSI_TO_MPA 						: REAL := 0.00689475729;
	MPA_TO_PSI						: REAL := 145.0377;
	FT3_TO_M3						: REAL := 1/35.3146662127;	//ft^3 to m^3
	M3_TO_FT3						: REAL := 35.3146662127;	//m^3 to ft^3
	SECONDS_IN_MINUTE				: REAL := 60;
	PERCENT_PER_DECIMAL				: REAL := 100;
	GAL_TO_L						: REAL := 3.78541;			//Gallons to Liters
	L_TO_GAL						: REAL := 0.264172;
	MILLI_PER_SECOND				: DINT := 1000;	
	MILLI_PER_MINUTE				: DINT := 60000;
	MILLI_PER_HOUR					: DINT := 3600000;
	LB_TO_DaN						: REAL := 0.444822;
	DaN_TO_LB						: REAL := 2.248089;
	LB_TO_KG						: REAL := 0.453592;
	KG_TO_LB						: REAL := 2.20462;
	FT_TO_M							: REAL := 0.3048;
	M_TO_FT							: REAL := 3.280839895;
	REAL_MAX						: REAL := 3.40282346E+38;
	REAL_MIN						: REAL := 1.179435E-38;
	IN3_TO_GAL						: REAL := 1/231.0;
	SCF_PER_GAL						: REAL := 93.11;			//Standard Cubic Ft (at 1 atm and 70°F) per Gallon of Liquid Nitrogen (LN2)
	PI								: REAL := 3.14159;
	KPA_TO_PSI						: REAL := 0.145038;			

END_VAR

// Version/Global_Version
{attribute 'TcGenerated'}
{attribute 'no-analysis'}
{attribute 'linkalways'}
// This function has been automatically generated from the project information.
VAR_GLOBAL CONSTANT
	{attribute 'const_non_replaced'}
	stLibVersion_stdNOV : ST_LibVersion := (iMajor := 1, iMinor := 0, iBuild := 0, iRevision := 2936, nFlags := 0, sVersion := '1.0.0.2936');
END_VAR

// 20 Program Organization Units/Alarms/f_AlarmCode
(*AUTHOR:			Jaison Schaab*)
(*DATE:				January 21 / 2020*)
(*DESCRIPTION: 		This Function will compose an alarm code from input
					device Id and fault code.*)
(*INPUTS:			devId		-	device Id
					code		-	fault code*)
(*OUTPUTS:			UAlarmCode	-	composed alarm code*)

(*NOTES:			
*)

(*UPDATE: 			March. 22 2021 - Jaison Schaab

					Code Is fully tested and functional.
					
*)

FUNCTION f_AlarmCode : UAlarmCode
VAR_INPUT
	devId	: UDeviceId;
	code	: UFaultCode;
END_VAR
VAR
END_VAR

f_AlarmCode.code.devId.devId 			:= devId.devId;
f_AlarmCode.code.faultCode.faultcode 	:= code.faultcode;

END_FUNCTION

// 20 Program Organization Units/Alarms/f_DeviceId
(*AUTHOR:			Jaison Schaab*)
(*DATE:				January 21 / 2020*)
(*DESCRIPTION: 		This Function will compose a device Id from input
					component Id and element Id.*)
(*INPUTS:			compId		-	component Id
					elemId		-	element Id*)
(*OUTPUTS:			UDeviceId	-	composed device Id*)

(*NOTES:			
*)

(*UPDATE: 			March. 22 2021 - Jaison Schaab

					Code Is fully tested and functional.
					
*)

FUNCTION f_DeviceId : UDeviceId
VAR_INPUT
	compId	: TComponentId;
	elemId	: TElementId;
END_VAR
VAR
END_VAR

f_DeviceId.devId.component 	:= compId;
f_DeviceId.devId.element 	:= elemId;

END_FUNCTION

// 20 Program Organization Units/Alarms/f_FaultCode
(*AUTHOR:			Jaison Schaab*)
(*DATE:				January 21 / 2020*)
(*DESCRIPTION: 		This Function will compose a fault code from input
					fault priority and fault condition.*)
(*INPUTS:			priority	-	fault priority
					condition	-	fault condition*)
					
(*OUTPUTS:			UFaultCode	-	composed fault code*)

(*NOTES:			
*)

(*UPDATE: 			March. 22 2021 - Jaison Schaab

					Code Is fully tested and functional.
					
*)

FUNCTION f_FaultCode : UFaultCode
VAR_INPUT
	priority	: TFaultPriority;
	condition	: TFaultCondition;
END_VAR
VAR
END_VAR

f_FaultCode.faultcode.priority 	:= priority;
f_FaultCode.faultcode.condition := condition;

END_FUNCTION

// 20 Program Organization Units/Alarms/f_GetFaultCodePriority
(*AUTHOR:			Jaison Schaab*)
(*DATE:				January 21 / 2020*)
(*DESCRIPTION: 		This Function will decode and return the priority number 
					for a given fault code input.*)
(*INPUTS:			code	-	fault code*)
(*OUTPUTS:			UINT	-	priority value of the fault code*)

(*NOTES:			This routine was written and intended to be used for
					the purpose of sorting the alarm list by priority.
*)

(*UPDATE: 			March. 22 2021 - Jaison Schaab

					Code Is fully tested and functional.
					
*)

FUNCTION f_GetFaultCodePriority : UINT
VAR_INPUT
	code	: UFaultCode;
END_VAR
VAR
END_VAR

f_GetFaultCodePriority := TO_UINT(SHR((code.faultcode_WORD AND 16#FF00), 8));

END_FUNCTION

// 20 Program Organization Units/Alarms/fb_AlarmHandler
(*AUTHOR:			Jaison Schaab*)
(*DATE:				December 30 / 2019*)
(*DESCRIPTION: 		This Function Block contains the alarm list and all methods
					to interact with it; including Set and Clear.*)
					
(*NOTES:			The alarm list is a static array which contains "_ALARM_ARRAY_MAX_SIZE"
					number of elements, however, not all will be populated.  When the Init
					method is called the alarm list will be initialized with ONLY those alarms
					which have text associated with them.  Use the GetNumOfAlarms method which
					returns the number of configured alarms.  If a SET or CLEAR method is 
					called on a non-existent alarm it will simply be ignored.
*)

(*UPDATE: 			March. 22 2021 - Jaison Schaab

					Code Is fully tested and functional.
					
					A fix had to be made in the "Init" method to pass the alarm message array in as a pointer
					instead of static array.  Beckhoff support is unsure why this was generating a TCOM error,
					however using a pointer fixed the issue and is a more efficient method of passing the array.
					
*)

(*UPDATE: 			March. 18 2021 - Jaison Schaab

					Code Ported from Wago.
					
					Code is NOT YET Operational. There is an issue with sharing memory from within a library
					that is not handled on the beckhoff which could be due to Beckhoff using an older version
					of Codesys from Wago.
*)

(*UPDATE: 			June. 23 2020 - Jaison Schaab

					Added "RegisterAlarmCode" function as well as 6 lists which track all of the
					availible registered alarm codes within the project.  These lists are as 
					follows:
						
						- m_RegAlarmCodeList - List of TAlarmCode
						- m_RegAlarmCodeDWORDList - List of DWORD;
						- m_RegDeviceComponentIdList - List of TComponentId;
						- m_RegDeviceElementIdList - List of TElementId;
						- m_RegFaultPriorityIdList - List of TFaultPriority;
						- m_RegFaultConditionIdList - List of TFaultCondition;
*)

FUNCTION_BLOCK fb_AlarmHandler
VAR_INPUT
END_VAR
VAR_OUTPUT
END_VAR
VAR
	// List of defined alarm codes, states, and messages
	m_alarmList					: ARRAY[0.._ALARM_ARRAY_MAX_SIZE] OF TAlarmType;
	
	m_numAlarms					: UINT;
	m_numActiveAlarms			: UINT;
	
	// Lists of all registered possible alarm codes
	m_RegAlarmCodeList			: ARRAY[1.._ALARM_ARRAY_MAX_SIZE + 1] OF TAlarmCode;
	m_RegAlarmCodeDWORDList		: ARRAY[1.._ALARM_ARRAY_MAX_SIZE + 1] OF DWORD;
	m_RegDeviceComponentIdList	: ARRAY[1.._ALARM_ARRAY_MAX_SIZE + 1] OF TComponentId;
	m_RegDeviceElementIdList	: ARRAY[1.._ALARM_ARRAY_MAX_SIZE + 1] OF TElementId;
	m_RegFaultPriorityIdList	: ARRAY[1.._ALARM_ARRAY_MAX_SIZE + 1] OF TFaultPriority;
	m_RegFaultConditionIdList	: ARRAY[1.._ALARM_ARRAY_MAX_SIZE + 1] OF TFaultCondition;
	
	m_numRegCodes				: UINT;
END_VAR

(* ---------------------------------------------------------------------------
Func name   : 	Clear
Description : 	Clears the state of the input alarm code if it is found
				in the alarm list, also updates the active alarm counter.
Inputs      :	code	- 	alarm code
Returns     : 	None
Notes       : 	
--------------------------------------------------------------------------- *)

METHOD Clear
VAR_INPUT
	code	: UAlarmCode;	// Input alarm code
END_VAR
VAR
	i		: UINT;			// Alarm list index
END_VAR
// Find the specified alarm in the alarm list
i := 0;

WHILE ((i < m_numAlarms) AND (m_alarmList[i].code.code_UDINT <> code.code_UDINT)) DO
	// Incriment to the next alarm message
	i := i + 1;	
END_WHILE

// If the alarm was found and active clear it.
IF ((i < m_numAlarms) AND (m_alarmList[i].state = TRUE)) THEN
	
	// Clear the alarm flag in the alarm list (static map)
	m_alarmList[i].state := FALSE;
	
	// Subtract alarm count from the active alarms
	m_numActiveAlarms := m_numActiveAlarms - 1;

END_IF
END_METHOD

(* ---------------------------------------------------------------------------
Func name   : 	FB_exit
Description : 	Destructor
Inputs      :	None
Returns     : 	None
Notes       : 	
--------------------------------------------------------------------------- *)

METHOD FB_exit
VAR_INPUT
	bInCopyCode : BOOL; // if TRUE, the exit method is called for exiting an instance that is copied afterwards (online change)
END_VAR
// Do nothing
END_METHOD

(* ---------------------------------------------------------------------------
Func name   : 	FB_init
Description : 	Constructor
Inputs      :	None
Returns     : 	None
Notes       : 	
--------------------------------------------------------------------------- *)

METHOD FB_init
VAR_INPUT
	bInitRetains 		: BOOL; // if TRUE, the retain variables are initialized (warm start / cold start)
    bInCopyCode  		: BOOL; // if TRUE, the instance afterwards gets moved into the copy code (online change)
END_VAR
m_numRegCodes := 0;
END_METHOD

(* ---------------------------------------------------------------------------
Func name   : 	GetAlarmCodeIndex
Description : 	Searches the internal alarm list and returns the
				array index of the specified alarm code.
Inputs      :	code	- 	alarm code
Returns     : 	UINT	- 	array index of alarm code
Notes       : 	
--------------------------------------------------------------------------- *)

METHOD GetAlarmCodeIndex : UINT
VAR_INPUT
	code	: UAlarmCode;	// Input alarm code
END_VAR
VAR		
	i		: INT;			// Alarm list index
END_VAR
// Find the specified alarm in the alarm list
i := 0;

// Stop searching once the desired Alarm Code is reached OR the end of the alarm list is found. <JAISON>
WHILE ((i < TO_INT(m_numAlarms)) AND (m_alarmList[i].code.code_UDINT <> code.code_UDINT)) DO
	
	// Incriment to the next alarm message
	i := i + 1;	
END_WHILE

GetAlarmCodeIndex := TO_UINT(i);
END_METHOD

(* ---------------------------------------------------------------------------
Func name   : 	GetAlarms
Description : 	Returns a pointer to the alarm list.
Inputs      :	None
Returns     : 	POINTER TO ARRAY[0.._ALARM_ARRAY_MAX_SIZE] OF AlarmType
Notes       : 	
--------------------------------------------------------------------------- *)

METHOD GetAlarms : POINTER TO ARRAY[0.._ALARM_ARRAY_MAX_SIZE] OF TAlarmType;
VAR_INPUT
END_VAR
GetAlarms := ADR(m_alarmList);
END_METHOD

(* ---------------------------------------------------------------------------
Func name   : 	GetNumOfActiveAlarms
Description : 	Retrieves the number of active alarms in the alarm list.
Inputs      :	None
Returns     : 	UINT	-	the number of active alarms
Notes       : 	
--------------------------------------------------------------------------- *)

METHOD GetNumOfActiveAlarms : UINT
VAR_INPUT
END_VAR
GetNumOfActiveAlarms := m_numActiveAlarms;
END_METHOD

(* ---------------------------------------------------------------------------
Func name   : 	GetNumOfAlarms
Description : 	Retrieves the number of configured alarms in the alarm list.
Inputs      :	None
Returns     : 	UINT	-	the number of alarms in the alarm list
Notes       : 	
--------------------------------------------------------------------------- *)

METHOD GetNumOfAlarms : UINT
VAR_INPUT
END_VAR
GetNumOfAlarms := m_numAlarms;
END_METHOD

(* ---------------------------------------------------------------------------
Func name   : 	GetNumOfDeviceId
Description : 	Searches the internal alarm list and returns the number of
				defined alarms with the input device id.
Inputs      :	devId		- 	input device id
Returns     : 	UINT		- 	the number of alarms with the input
								device id in the alarm list
Notes       : 	
--------------------------------------------------------------------------- *)

METHOD GetNumOfDeviceId : UINT
VAR_INPUT
	devId	: UDeviceId;	// Input device id
END_VAR
VAR		
	i		: INT;
	num		: UINT;
END_VAR
// Find the specified alarm in the alarm list
i := 0;
num := 0;

// Stop searching once the desired DeviceId is reached OR the end of the alarm list is found.
// This can be done because we know the alarm list is sorted from lowest to highest device ID. <JAISON>
WHILE ((i < TO_INT(m_numAlarms)) AND (m_alarmList[i].code.code.devId.devId_UINT <= devId.devId_UINT)) DO
	
	IF (m_alarmList[i].code.code.devId.devId_UINT = devId.devId_UINT) THEN
		num := num + 1;
	END_IF
	
	// Incriment to the next alarm message
	i := i + 1;	
END_WHILE

GetNumOfDeviceId := num;
END_METHOD

(* ---------------------------------------------------------------------------
Func name   : 	GetNumRegisteredCodes
Description : 	Retrieves the number of registered alarm codes in the project.
Inputs      :	None
Returns     : 	UINT	-	the number of registered alarm codes
Notes       : 	
--------------------------------------------------------------------------- *)

METHOD GetNumRegisteredCodes : UINT
VAR_INPUT
END_VAR
GetNumRegisteredCodes := m_numRegCodes;
END_METHOD

(* ---------------------------------------------------------------------------
Func name   : 	GetRegisteredAlarmCodeDWORDListPointer
Description : 	Returns a pointer to the registered alarm code list. 
Inputs      :	None
Returns     : 	POINTER TO ARRAY[1.._ALARM_ARRAY_MAX_SIZE + 1] OF DWORD
Notes       : 	
--------------------------------------------------------------------------- *)

METHOD GetRegisteredAlarmCodeDWORDListPointer : POINTER TO ARRAY[1.._ALARM_ARRAY_MAX_SIZE + 1] OF DWORD
VAR_INPUT
END_VAR
GetRegisteredAlarmCodeDWORDListPointer := ADR(m_RegAlarmCodeDWORDList);
END_METHOD

(* ---------------------------------------------------------------------------
Func name   : 	GetRegisteredAlarmCodeListPointer
Description : 	Returns a pointer to the registered alarm code list. 
Inputs      :	None
Returns     : 	POINTER TO ARRAY[1.._ALARM_ARRAY_MAX_SIZE + 1] OF TAlarmCode
Notes       : 	
--------------------------------------------------------------------------- *)

METHOD GetRegisteredAlarmCodeListPointer : POINTER TO ARRAY[1.._ALARM_ARRAY_MAX_SIZE + 1] OF TAlarmCode
VAR_INPUT
END_VAR
GetRegisteredAlarmCodeListPointer := ADR(m_RegAlarmCodeList);
END_METHOD

(* ---------------------------------------------------------------------------
Func name   : 	GetRegisteredDeviceComponentIdListPointer
Description : 	Returns a pointer to the registered device component Id list. 
Inputs      :	None
Returns     : 	POINTER TO ARRAY[1.._ALARM_ARRAY_MAX_SIZE + 1] OF TComponentId
Notes       : 	
--------------------------------------------------------------------------- *)

METHOD GetRegisteredDeviceComponentIdListPointer : POINTER TO ARRAY[1.._ALARM_ARRAY_MAX_SIZE + 1] OF TComponentId;
VAR_INPUT
END_VAR
GetRegisteredDeviceComponentIdListPointer := ADR(m_RegDeviceComponentIdList);
END_METHOD

(* ---------------------------------------------------------------------------
Func name   : 	GetRegisteredDeviceElementIdListPointer
Description : 	Returns a pointer to the registered device element Id list. 
Inputs      :	None
Returns     : 	POINTER TO ARRAY[1.._ALARM_ARRAY_MAX_SIZE + 1] OF TElementId
Notes       : 	
--------------------------------------------------------------------------- *)

METHOD GetRegisteredDeviceElementIdListPointer : POINTER TO ARRAY[1.._ALARM_ARRAY_MAX_SIZE + 1] OF TElementId;
VAR_INPUT
END_VAR
GetRegisteredDeviceElementIdListPointer := ADR(m_RegDeviceElementIdList);
END_METHOD

(* ---------------------------------------------------------------------------
Func name   : 	GetRegisteredFaultCondiitionIdListPointer
Description : 	Returns a pointer to the registered fault condition Id list. 
Inputs      :	None
Returns     : 	POINTER TO ARRAY[1.._ALARM_ARRAY_MAX_SIZE + 1] OF TFaultCondition
Notes       : 	
--------------------------------------------------------------------------- *)

METHOD GetRegisteredFaultCondiitionIdListPointer : POINTER TO ARRAY[1.._ALARM_ARRAY_MAX_SIZE + 1] OF TFaultCondition;
VAR_INPUT
END_VAR
GetRegisteredFaultCondiitionIdListPointer := ADR(m_RegFaultConditionIdList);
END_METHOD

(* ---------------------------------------------------------------------------
Func name   : 	GetRegisteredFaultPriorityIdListPointer
Description : 	Returns a pointer to the registered fault priority Id list. 
Inputs      :	None
Returns     : 	POINTER TO ARRAY[1.._ALARM_ARRAY_MAX_SIZE + 1] OF TFaultPriority
Notes       : 	
--------------------------------------------------------------------------- *)

METHOD GetRegisteredFaultPriorityIdListPointer : POINTER TO ARRAY[1.._ALARM_ARRAY_MAX_SIZE + 1] OF TFaultPriority;
VAR_INPUT
END_VAR
GetRegisteredFaultPriorityIdListPointer := ADR(m_RegFaultPriorityIdList);
END_METHOD

(* ---------------------------------------------------------------------------
Func name   : 	Init
Description : 	Initializes the alarm list which will comprise of all elements
				that exist in the input alarm message array.  The internal array
				is then sorted by priority from lowest to highest.
Inputs      :	pAlarmMsg	-	pointer to the static array of alarm messages
Returns     : 	None
Notes       : 	This method is done outside the FB_Init constructor
				because the alarm handler is defined in global memory,
				but needs to be initialized by the alarm interface.
--------------------------------------------------------------------------- *)

(*UPDATE: 			April. 16 2020 - Jaison Schaab

					Added a check before the bubble sort to ensure that the
					number of configured alarms is greater than 1.  Otherwise,
					the code will cause memory errors.*)

METHOD Init
VAR_INPUT
	pAlarmMsg		: POINTER TO ARRAY[0.._ALARM_ARRAY_MAX_SIZE] OF TAlarmMessage;	// Static array of alarm messages pointer
END_VAR
VAR
	i				: UINT;			// Alarm list index
	j				: UINT;			// Bubble sort alarm list index
	temp			: TAlarmType;	// Bubble sort swap variable
END_VAR
// Associate alarm messages to the alarm codes. The 'alarmMsg' array is a pre-defined
// static array.  Use the code being 0 define the end of the defined array.
i := 0;
WHILE ((pAlarmMsg^[i].code.code_DWORD > 0) AND (i < _ALARM_ARRAY_MAX_SIZE)) DO
	
	m_alarmList[i].code := pAlarmMsg^[i].code;
	m_alarmList[i].state := FALSE;
	m_alarmList[i].message := pAlarmMsg^[i].msg;

	// Incriment to the next alarm message
	i := i + 1;	
END_WHILE

m_numAlarms := i;

// Sort the alarm array by alarm code value from lowest to highest
// using a bubble sort algorithm. <JAISON>
//
// O(n*n) 	Worst and Average Case Time Complexity
//			Worst case occurs when array is reverse sorted
//
// O(n)		Best Case Time Complexity
//			Best case occurs when array is already sorted

IF (m_numAlarms > 1) THEN
	
	FOR i:=0 TO m_numAlarms - 1 BY 1 DO
		
		FOR j:=0 TO m_numAlarms - 1 - 1 BY 1 DO
			
			IF (m_alarmList[j].code.code_UDINT > m_alarmList[j+1].code.code_UDINT) THEN
				
				temp := m_alarmList[j+1];
				
				m_alarmList[j+1] := m_alarmList[j];
				
				m_alarmList[j] := temp;			
			
			END_IF
		
		END_FOR
		
	END_FOR;
	
END_IF
END_METHOD

(* ---------------------------------------------------------------------------
Func name   : 	RegisterAlarmCode
Description : 	Registers input alarm code to the various lists and also 
				updates the number of registered code counter.
Inputs      :	code	- 	alarm code
Returns     : 	None
Notes       : 	Every function that can sets a fault in the alarm handler
				is responsible for registering the code with this function.
				
				To make it easier, it is best to use the fb_AlarmMonitor
				interface as it will register the code here automatically.
--------------------------------------------------------------------------- *)

METHOD RegisterAlarmCode
VAR_INPUT
	code	: UAlarmCode;	// Input alarm code
END_VAR
// Add the registered alarm code to the lists for tracking
m_RegAlarmCodeList[m_numRegCodes + 1] 			:= code.code;
m_RegAlarmCodeDWORDList[m_numRegCodes + 1] 		:= code.code_DWORD;
m_RegDeviceComponentIdList[m_numRegCodes + 1]	:= code.code.devId.devId.component;
m_RegDeviceElementIdList[m_numRegCodes + 1]		:= code.code.devId.devId.element;
m_RegFaultPriorityIdList[m_numRegCodes + 1]		:= code.code.faultCode.faultcode.priority;
m_RegFaultConditionIdList[m_numRegCodes + 1]	:= code.code.faultCode.faultcode.condition;

// Increment the number of registered codes to keep track of the total defined in the project
m_numRegCodes := m_numRegCodes + 1;
END_METHOD

(* ---------------------------------------------------------------------------
Func name   : 	Set
Description : 	Sets the state of the input alarm code if it is found
				in the alarm list, also updates the active alarm counter.
Inputs      :	code	- 	alarm code
Returns     : 	None
Notes       : 	
--------------------------------------------------------------------------- *)

METHOD Set
VAR_INPUT
	code	: UAlarmCode;	// Input alarm code
END_VAR
VAR		
	i		: UINT;			// Alarm list index
END_VAR
// Find the specified alarm in the alarm list
i := 0;

WHILE ((i < m_numAlarms) AND (m_alarmList[i].code.code_UDINT <> code.code_UDINT)) DO
	// Incriment to the next alarm message
	i := i + 1;	
END_WHILE

// If the alarm was found and not active set it.
IF ((i < m_numAlarms) AND (m_alarmList[i].state = FALSE)) THEN
	
	// Set the alarm flag in the alarm list (static map)
	m_alarmList[i].state := TRUE;
	
	// Add alarm count to the active alarms
	m_numActiveAlarms := m_numActiveAlarms + 1;	
		
END_IF
END_METHOD

END_FUNCTION_BLOCK

// 20 Program Organization Units/Alarms/fb_AlarmMonitor
(*AUTHOR:			Jaison Schaab*)
(*DATE:				January 20 / 2020*)
(*DESCRIPTION: 		This Function Block provides a standard interface into the alarm handler
					where a user can set limits, either INT, REAL or BOOL and pass in a 
					variable to be monitored based on those limits.*)

			
(*NOTES:			User MUST call a set limit method (SetLimitBool, SetLimit,Int,
					SetLimitReal) and also enable the limits using the EnableLimit
					method prior to calling a monitor method (MonitorBool, MonitorInt,
					MonitorReal).
*)

(*UPDATE: 			March. 22 2021 - Jaison Schaab

					Code Is fully tested and functional.
					
*)

(*UPDATE: 			March. 18 2021 - Jaison Schaab

					Code Ported from Wago.
					
					Code is NOT YET Operational. There is an issue with sharing memory from within a library
					that is not handled on the beckhoff which could be due to Beckhoff using an older version
					of Codesys from Wago.
*)

(*UPDATE: 			February. 7 2020 - Jaison Schaab

					Added a "monitorType" to the TAlarmLimit data type which will track whether this
					instantiation of the alarm monitor is an "upper_limit" or "lower_limit" type.
					Having to verbosly specify this rather than deduce this from the input on/off values
					ensures that the operator is aware of what conditions are being monitored as well as
					allows error checking in the SetLimit routines.

					The SetLimit routines will now return a BOOL indicating whether they worked or not based
					on the validity of the values passed in.
						
					This change affects the following methods of the fb_AlarmMonitor:
					
						- FB_Init
						- Monitor
						- MonitorBool
						- MonitorInt
						- MonitorReal
						- SetLimitBool
						- SetLimitInt
						- SetLimitReal
*)

(*UPDATE: 			June. 23 2020 - Jaison Schaab

					Added "m_pAlarmHandler^.RegisterAlarmCode" function calls in the InitAlarms Method which is required to
					populate the registered alarm code lists in the fb_AlarmHandler class.		
*)

FUNCTION_BLOCK fb_AlarmMonitor
VAR_INPUT

END_VAR
VAR_OUTPUT

END_VAR
VAR
	m_code				: UAlarmCode;					// Alarm code associated with the monitor
	m_initialized		: BOOL;							// Monitor initialization flag (TRUE = initialized)
	
	m_limit				: TAlarmLimit;					// Limit (on value, off value, enable, monitor type)
	
	m_limitOnTON		: TON;							// Timer ON for alarm set delay
	m_limitOn			: R_TRIG;						// Positive edge detection (set alarm)
	m_limitOff			: F_TRIG;						// Negative edge detection (clear alarm)
	
	m_state				: BOOL;
	m_pAlarmHandler		: POINTER TO fb_AlarmHandler;	// Alarm handler function pointer
END_VAR

(* ---------------------------------------------------------------------------
Func name   : 	CheckLimits
Description : 	Checks the input limits to ensure they match the defined monitor
				type (ie. if configured as a "lower_limit" then the ON value
				should be LESS THAN or EQUAL TO the OFF value).
Inputs      :	on		- 	alarm limit ON value 
				off		- 	alarm limit OFF value
Returns     : 	BOOL	-	TRUE on success, else FALSE
Notes       : 	This routine uses an LREAL value format.  This was decided
				as the generic type used as it can encompass any particular
				types needed to be monitored.  All monitor routines can simply
				convert their values to LREAL (64 bit) and call this routine.
--------------------------------------------------------------------------- *)

METHOD CheckLimits : BOOL
VAR_INPUT
	on	: LREAL;	// Value which SETS the alarm
	off	: LREAL;	// Value which CLEARS the alarm
END_VAR
// If the monitor is NOT yet initialized allow the SETTING of the 
// values as they will be from the constructor which is run before
// InitAlarms which is where the monitor is given its type. <JAISON>
IF (m_initialized) THEN

	CASE m_limit.monitorType OF
	TAlarmMonitorType.lower_limit:	// Lower Limit monitor type defined
	
		// A lower limit range will have an 'on' value less than or equal to the 'off' value
		IF (on <= off) THEN
			CheckLimits := TRUE;
		ELSE
			CheckLimits := FALSE;
		END_IF
	
	TAlarmMonitorType.upper_limit:	// Upper Limit monitor type defined
	
		// A upper limit range will have an 'on' value greater than or equal to the 'off' value
		IF (on >= off) THEN
			CheckLimits := TRUE;
		ELSE
			CheckLimits := FALSE;
		END_IF
	
	ELSE							// Unknown monitor type error - Return FALSE
		
		CheckLimits := FALSE;
		
	END_CASE;
	
ELSE
	CheckLimits := TRUE;
END_IF
END_METHOD

(* ---------------------------------------------------------------------------
Func name   : 	DisableLimit
Description : 	Deactivates the monitoring routine.
Inputs      :	None
Returns     : 	None
Notes       : 	This method will also clear an active alarm if it exists.
--------------------------------------------------------------------------- *)

METHOD DisableLimit
VAR_INPUT
END_VAR
IF (m_limit.enable) THEN
	m_limit.enable := FALSE;			// inactive
	m_pAlarmHandler^.Clear(m_code);		// clear alarm if it was already active
END_IF
END_METHOD

(* ---------------------------------------------------------------------------
Func name   : 	EnableLimit
Description : 	Activates the alarm monitor routine.
Inputs      :	None
Returns     : 	None
Notes       : 	
--------------------------------------------------------------------------- *)

METHOD EnableLimit
VAR_INPUT
END_VAR
m_limitOn(CLK:= FALSE);				// set FALSE to detect if alarm is already active
m_limitOnTON(IN:= FALSE);			// reset the ON delay timer
m_limit.enable := TRUE;				// active
END_METHOD

(* ---------------------------------------------------------------------------
Func name   : 	FB_exit
Description : 	Destructor
Inputs      :	None
Returns     : 	None
Notes       : 	
--------------------------------------------------------------------------- *)

METHOD FB_exit
VAR_INPUT
	bInCopyCode : BOOL; // if TRUE, the exit method is called for exiting an instance that is copied afterwards (online change)
END_VAR
// Do nothing
END_METHOD

(* ---------------------------------------------------------------------------
Func name   : 	FB_init
Description : 	Constructor
Inputs      :	None
Returns     : 	None
Notes       : 	
--------------------------------------------------------------------------- *)

METHOD FB_init
VAR_INPUT
	bInitRetains 		: BOOL; 				// if TRUE, the retain variables are initialized (warm start / cold start)
    bInCopyCode  		: BOOL; 				// if TRUE, the instance afterwards gets moved into the copy code (online change)
END_VAR
// Ensure initialization flag is false so user MUST call init function
// which will set the alarm code and delay time variables <JAISON>
m_initialized := FALSE;

// Set the local alarm handler pointer to the global handler
m_pAlarmHandler := ADR(gAlarmHandler);

// Initialize the 'limitOn' positive edge detect signal to low so that
// we detect a positive edge if the signal is high at startup.
m_limitOn(CLK:= FALSE);

// Disable the limits initially
m_limit.enable := FALSE;
m_limit.limitOn := 0;
m_limit.limitOff := 0;
END_METHOD

METHOD GetState : BOOL
VAR_INPUT
END_VAR
GetState := m_state;
END_METHOD

(* ---------------------------------------------------------------------------
Func name   : 	InitAlarm
Description : 	Initialization routine required to set the alarm code associated
				with the monitor, as well as the delay time.
Inputs      :	code		-	alarm code associated with the monitor
				delayTime	-	alarm set delay time
Returns     : 	None
Notes       : 	
--------------------------------------------------------------------------- *)

METHOD InitAlarm
VAR_INPUT	
	code			: UAlarmCode; 			// Alarm code consisting of the DeviceId and FaultCode associated with the monitor
	alarmType		: TAlarmMonitorType;		// Alarm monitor type which indicates whether this is a 
	delayTime		: TIME;					// Delay time for setting the alarm used to prevent false alarm trips
END_VAR
// Set the alarm code
m_code := code;

// Set the timer default value
m_limitOnTON.PT := delayTime;

// Set the local alarm handler pointer to the global handler
m_pAlarmHandler := ADR(gAlarmHandler);

// Initialize the 'limitOn' positive edge detect signal to low so that
// we detect a positive edge if the signal is high at startup.
m_limitOn(CLK:= FALSE);

// Disable the limits initially
m_limit.enable := FALSE;
m_limit.limitOn := 0;
m_limit.limitOff := 0;
m_limit.monitorType := alarmType;

// Set the initialization flag
m_initialized := TRUE;

// Register the handled alarm codes
m_pAlarmHandler^.RegisterAlarmCode(code);
END_METHOD

(* ---------------------------------------------------------------------------
Func name   : 	Monitor
Description : 	Common monitor routine which will handle both upper and lower
				limit monitoring of an input value using preset ON and OFF
				limit values (passed in constructor).  This routine also
				utilizes an ON delay timer to prevent false trips.
Inputs      :	value	- 	value to me monitored
Returns     : 	BOOL	-	TRUE on success, else FALSE
Notes       : 	This routine will handle both the case when the ON value is
				greater then the OFF value and also if the OFF value is greater
				than or equal to the ON value based on input monitor type.

				This routine uses an LREAL value format.  This was decided
				as the generic type used as it can encompass any particular
				types needed to be monitored.  All monitor routines can simply
				convert their values to LREAL (64 bit) and call this routine.
--------------------------------------------------------------------------- *)

METHOD PRIVATE Monitor : BOOL
VAR_INPUT
	value		: LREAL;	// value to be monitored in generic LREAL format
END_VAR
// ONLY monitor if the Init routine has been run
IF (m_initialized) THEN
	
	// Check the state (active/inactive)
	IF (m_limit.enable) THEN
		
		// A lower limit range will have an 'on' value less than the 'off' value
		//IF (m_limit.limitOn < m_limit.limitOff) THEN
		IF (m_limit.monitorType = TAlarmMonitorType.lower_limit) THEN
			
			// Lower limit check
	
			// Use a TON delay timer
			m_limitOnTON(IN:= (value <= m_limit.limitOn));
	
			// Set an alarm condition on the positive edge
			m_limitOn(CLK:= m_limitOnTON.Q);
			IF (m_limitOn.Q) THEN
				
				// Set the alarm
				m_pAlarmHandler^.Set(m_code);
				m_state := TRUE;
			END_IF
	
			// Clear the alarm condition on a negative edge
			m_limitOff(CLK:= (value < m_limit.limitOff));
			IF (m_limitOff.Q) THEN
				
				// Clear the alarm
				m_pAlarmHandler^.Clear(m_code);
				m_state := FALSE;
			END_IF	
	
		// A upper limit range will have an 'on' value greater than the 'off' value
		ELSIF (m_limit.monitorType = TAlarmMonitorType.upper_limit) THEN
			
			// Upper limit check
	
			// Use a TON delay timer
			m_limitOnTON(IN:= (value >= m_limit.limitOn));
	
			// Set an alarm condition on the positive edge
			m_limitOn(CLK:= m_limitOnTON.Q);
			IF (m_limitOn.Q) THEN
				
				// Set the alarm
				m_pAlarmHandler^.Set(m_code);
				m_state := TRUE;
			END_IF
	
			// Clear the alarm condition on a negative edge
			m_limitOff(CLK:= (value > m_limit.limitOff));
			IF (m_limitOff.Q) THEN
				
				// Clear the alarm
				m_pAlarmHandler^.Clear(m_code);
				m_state := FALSE;
			END_IF
		
			// Monitor is initialized and running
			Monitor := TRUE;
			
		ELSE
			
			// Monitor Type is Invalid
			Monitor := FALSE;
				
		END_IF
	
	ELSE

		// Limit is Disabled	
		Monitor := FALSE;
		
	END_IF
	
	// Monitor is Disabled
	Monitor := FALSE;
	
END_IF
END_METHOD

(* ---------------------------------------------------------------------------
Func name   : 	MonitorBool
Description : 	Monitors a BOOL input value against preset limits to set
				and clear the alarm represented by the alarm code in the
				alarm list.
Inputs      :	value	- 	value to me monitored
Returns     : 	BOOL	-	TRUE on success, else FALSE
Notes       : 	Input value is simply converted to a generic LREAL
				format and passed to common monitor routine.
--------------------------------------------------------------------------- *)

METHOD MonitorBool : BOOL
VAR_INPUT
	value		: BOOL;
END_VAR
// Convert the input value to LREAL and pass to monitor routine
MonitorBool := Monitor(value:= BOOL_TO_LREAL(value));
END_METHOD

(* ---------------------------------------------------------------------------
Func name   : 	MonitorInt
Description : 	Monitors an INT input value against preset limits to set
				and clear the alarm represented by the alarm code in the
				alarm list.
Inputs      :	value	- 	value to me monitored
Returns     : 	BOOL	-	TRUE on success, else FALSE
Notes       : 	Input value is simply converted to a generic LREAL
				format and passed to common monitor routine.
--------------------------------------------------------------------------- *)

METHOD MonitorInt : BOOL
VAR_INPUT
	value		: INT;
END_VAR
// Convert the input value to LREAL and pass to monitor routine
MonitorInt := Monitor(value:= INT_TO_LREAL(value));
END_METHOD

(* ---------------------------------------------------------------------------
Func name   : 	MonitorReal
Description : 	Monitors a REAL input value against preset limits to set
				and clear the alarm represented by the alarm code in the
				alarm list.
Inputs      :	value	- 	value to me monitored
Returns     : 	BOOL	-	TRUE on success, else FALSE
Notes       : 	Input value is simply converted to a generic LREAL
				format and passed to common monitor routine.
--------------------------------------------------------------------------- *)

METHOD MonitorReal : BOOL
VAR_INPUT
	value		: REAL;
END_VAR
// Convert the input value to LREAL and pass to monitor routine
MonitorReal := Monitor(value:= REAL_TO_LREAL(value));
END_METHOD

(* ---------------------------------------------------------------------------
Func name   : 	SetDelayOn
Description : 	Sets the monitor on time delay value.
Inputs      :	delayTime	- 	alarm set delay time
Returns     : 	None
Notes       : 	
--------------------------------------------------------------------------- *)

METHOD SetDelayOn
VAR_INPUT
	delayTime	: TIME;		// Delay time for setting the alarm used to prevent false alarm trips
END_VAR
// Set the timer value
m_limitOnTON.PT := delayTime;
END_METHOD

(* ---------------------------------------------------------------------------
Func name   : 	SetLimitBool
Description : 	Sets the on/off limits for the alarm monitor routine
				in a BOOL format.
Inputs      :	on		- 	alarm limit ON value 
				off		- 	alarm limit OFF value
Returns     : 	BOOL	-	TRUE on success, else FALSE
Notes       : 	The limit values are stored in LREAL formats which was decided
				as the generic type used as it can encompass any particular
				types needed to be monitored.  All input types are simply
				converted to LREAL (64 bit) for comparison in the monitor.
--------------------------------------------------------------------------- *)

METHOD SetLimitBool : BOOL
VAR_INPUT
	on		: BOOL;		// Value which SETS the alarm
	off		: BOOL;		// Value which CLEARS the alarm
END_VAR
VAR
	m_on	: LREAL;	// internal converted ON value
	m_off	: LREAL;	// internal converted OFF value
END_VAR
// convert the inputs to LREAL for error checking
m_on := BOOL_TO_LREAL(on);
m_off := BOOL_TO_LREAL(off);

// Check that the limits match the configured alarm monitor type
IF (CheckLimits(on:= m_on, off:= m_off)) THEN

	// Limits are valid so update the parameters
	m_limit.limitOn := m_on;
	m_limit.limitOff := m_off;
	SetLimitBool := TRUE;

ELSE
	
	// Limits are invalid so ignore them
	SetLimitBool := FALSE;

END_IF
END_METHOD

(* ---------------------------------------------------------------------------
Func name   : 	SetLimitInt
Description : 	Sets the on/off limits for the alarm monitor routine
				in a INT format.
Inputs      :	on		- 	alarm limit ON value 
				off		- 	alarm limit OFF value
Returns     : 	BOOL	-	TRUE on success, else FALSE
Notes       : 	The limit values are stored in LREAL formats which was decided
				as the generic type used as it can encompass any particular
				types needed to be monitored.  All input types are simply
				converted to LREAL (64 bit) for comparison in the monitor.
--------------------------------------------------------------------------- *)

METHOD SetLimitInt : BOOL
VAR_INPUT
	on		: INT;		// Value which SETS the alarm
	off		: INT;		// Value which CLEARS the alarm
END_VAR
VAR
	m_on	: LREAL;	// internal converted ON value
	m_off	: LREAL;	// internal converted OFF value
END_VAR
// convert the inputs to LREAL for error checking
m_on := INT_TO_LREAL(on);
m_off := INT_TO_LREAL(off);

// Check that the limits match the configured alarm monitor type
IF (CheckLimits(on:= m_on, off:= m_off)) THEN

	// Limits are valid so update the parameters
	m_limit.limitOn := m_on;
	m_limit.limitOff := m_off;
	SetLimitInt := TRUE;

ELSE
	
	// Limits are invalid so ignore them
	SetLimitInt := FALSE;

END_IF
END_METHOD

(* ---------------------------------------------------------------------------
Func name   : 	SetLimitReal
Description : 	Sets the on/off limits for the alarm monitor routine
				in a REAL format.
Inputs      :	on		- 	alarm limit ON value 
				off		- 	alarm limit OFF value
Returns     : 	BOOL	-	TRUE on success, else FALSE
Notes       : 	The limit values are stored in LREAL formats which was decided
				as the generic type used as it can encompass any particular
				types needed to be monitored.  All input types are simply
				converted to LREAL (64 bit) for comparison in the monitor.
--------------------------------------------------------------------------- *)

METHOD SetLimitReal : BOOL
VAR_INPUT
	on		: REAL;		// Value which SETS the alarm
	off		: REAL;		// Value which CLEARS the alarm
END_VAR
VAR
	m_on	: LREAL;	// internal converted ON value
	m_off	: LREAL;	// internal converted OFF value
END_VAR
// convert the inputs to LREAL for error checking
m_on := REAL_TO_LREAL(on);
m_off := REAL_TO_LREAL(off);

// Check that the limits match the configured alarm monitor type
IF (CheckLimits(on:= m_on, off:= m_off)) THEN

	// Limits are valid so update the parameters
	m_limit.limitOn := m_on;
	m_limit.limitOff := m_off;
	SetLimitReal := TRUE;

ELSE
	
	// Limits are invalid so ignore them
	SetLimitReal := FALSE;

END_IF
END_METHOD

END_FUNCTION_BLOCK

// 20 Program Organization Units/Alarms/fb_AlarmInterface
(*AUTHOR:			Jaison Schaab*)
(*DATE:				January 20 / 2020*)
(*DESCRIPTION: 		This Function Block provides an interface into the alarm system, intended for
					integration with an HMI.  A pointer to a AlarmData structure memory space is
					provided which will be initialized and updated to match the internal alarm list.
					The AlarmData structure not only provides the alarm text, code and state but adds
					elements specific to the interface (Such as an ACK flag).*)

(*NOTES:			This function block and AlarmData structure was designed based on the legacy
					OPC Beijer alarm interface.  During the design of this system it has been determined
					that going forward this data structure is the best option; however, because the interface
					is abstracted away from the internal alarm list this interface can grow and change to meet
					any future interface needs.
					
					A future improvement which has been discussed is the inclusion of text (STRING) arrays 
					matching the FaultCode, ComponentId, and ElementId ENUMs in the interface.  This addition
					would allow the HMI or any device interfacing with the alarm system to decode the alarm codes
					and use them in some meaningful way.  In order to provide this functionality a second array
					containing the string definitions of each ENUM parameter would need to be added which creates
					double maintenance for the user/system designer.  Because the interfacing system currently does
					not require this it was decided to leave this out currently.
*)

(*UPDATE: 			March. 22 2021 - Jaison Schaab

					Code Is fully tested and functional.
					
					A fix had to be made in the "FB_Init" method to pass the alarm message array in as a pointer
					instead of static array.  Beckhoff support is unsure why this was generating a TCOM error,
					however using a pointer fixed the issue and is a more efficient method of passing the array.
					
*)

(*UPDATE: 			March. 18 2021 - Jaison Schaab

					Code Ported from Wago.
					
					Fixed an initial issue causing a TCOM error which prevented the code from running which
					was being caused by passing the TAlarmMessage array into the m_pAlarmHandler^.Init function
					within the FB_INIT method.  Apparently FB_INIT methods cannot pass data that way so as soon
					as I passed a pointer it worked.  This may be related to the issue below with the different
					memory (GUID) spaces between the library and mainline of code, I am not yet sure.  But making
					this change did NOT affect any operation and allows the code to run, albeit without any alarm
					data as the fb_AlarmHandler object is not being populated correctly.
					
					Code is NOT YET Operational. There is an issue with sharing memory from within a library
					that is not handled on the beckhoff which could be due to Beckhoff using an older version
					of Codesys from Wago.
					
*)

(*UPDATE: 			February. 7 2020 - Jaison Schaab
					Added the "AlarmState" to the AlarmData structure.  This state used by the HMI to 
					change the alarm icon depending on number of active alarms and their ack status.
					This variable tracks the following conditions for use on the HMI display:
					
						0 = Denotes NO active alarms present
						1 = Denotes active alarms present with ALL Acked
						2 = Denotes active alarms present AND AT LEAST 1 is NOT Acked
						
					This change affects ALL methods of the fb_AlarmInterface.*)

FUNCTION_BLOCK fb_AlarmInterface
VAR_INPUT
	xEnable						: BOOL;							// Function block enable - TRUE to enable
END_VAR
VAR_OUTPUT
	uiNumActiveAlarms			: UINT;							// Number of active alarms
END_VAR
VAR
	m_pAlarmHandler				: POINTER TO fb_AlarmHandler;	// Alarm handler function pointer
	m_pAlarmData				: POINTER TO TAlarmData;		// Interface alarm data structure pointer
	
	m_numAlarms					: UINT;							// Total number of configured alarms
	m_filterPriority			: BOOL;							// Filter (ignore) lower priority interface alarms when TRUE
	
	m_ResetTrigger				: F_TRIG;						// Falling edge trigger for enable input
END_VAR

IF (xEnable) THEN

	// Update the Interface Alarm Data each scan
	UpdateAlarms();

END_IF

// output the number of active system alarms
uiNumActiveAlarms := TO_UINT(m_pAlarmData^.NumOfActiveAlarms);

// Reset the alarm interface on enable input falling edge
m_ResetTrigger(CLK:= xEnable);

IF (m_ResetTrigger.Q) THEN
	ResetAlarms();
END_IF

(* ---------------------------------------------------------------------------
Func name   : 	FB_exit
Description : 	Destructor
Inputs      :	None
Returns     : 	None
Notes       : 	
--------------------------------------------------------------------------- *)

METHOD FB_exit
VAR_INPUT
	bInCopyCode : BOOL; // if TRUE, the exit method is called for exiting an instance that is copied afterwards (online change)
END_VAR
// Do nothing
END_METHOD

(* ---------------------------------------------------------------------------
Func name   : 	FB_init
Description : 	Constructor
Inputs      :	pAlarmMsg		-	pointer to the static array of alarm messages
				pAlarmData		-	pointer to the interface AlarmData structure
				xFilterPriority	-	filtering enable flag, TRUE to enable
Returns     : 	None
Notes       : 	
--------------------------------------------------------------------------- *)

METHOD FB_init
VAR_INPUT
	bInitRetains 	: BOOL; 														// if TRUE, the retain variables are initialized (warm start / cold start)
    bInCopyCode  	: BOOL; 														// if TRUE, the instance afterwards gets moved into the copy code (online change)
	pAlarmMsg		: POINTER TO ARRAY[0.._ALARM_ARRAY_MAX_SIZE] OF TAlarmMessage;	// Static array of alarm messages pointer
	pAlarmData		: POINTER TO TAlarmData;										// Interface Alarm data structure pointer
	xFilterPriority	: BOOL;															// Enable filtering (ignoring) of lower priority interface alarms when TRUE
END_VAR
VAR
	m_pAlarms		: POINTER TO ARRAY[0.._ALARM_ARRAY_MAX_SIZE] OF TAlarmType;	// Alarm Data
	
	i				: INT;														// Alarm list index
END_VAR
// Set the local alarm handler pointer to the global handler
m_pAlarmHandler := ADR(gAlarmHandler);

// Set the local alarm interface pointer
m_pAlarmData := pAlarmData;

// Initialize the Alarm Handler
m_pAlarmHandler^.Init(pAlarmMsg:= pAlarmMsg);

// Get the total number of configured alarms
m_numAlarms := m_pAlarmHandler^.GetNumOfAlarms();

// Set the filter priority flag
m_filterPriority := xFilterPriority;

// Get the system alarms list
m_pAlarms := m_pAlarmHandler^.GetAlarms();

// Iterate over the internal alarm list and add items to the interface alarm array
FOR i:=0 TO TO_INT(m_numAlarms) - 1 BY 1 DO
 
	// Initialize the Alarm Interface Array
	m_pAlarmData^.Alarm[i].code := m_pAlarms^[i].code.code_UDINT;
	m_pAlarmData^.Alarm[i].state := m_pAlarms^[i].state;
	m_pAlarmData^.Alarm[i].ack := FALSE;
	m_pAlarmData^.Alarm[i].message := m_pAlarms^[i].message;

END_FOR;

m_pAlarmData^.NumOfAlarms := TO_INT(m_numAlarms);
m_pAlarmData^.NumOfActiveAlarms := TO_INT(m_pAlarmHandler^.GetNumOfActiveAlarms());
m_pAlarmData^.RefreshAlarms := TRUE;	// Not sure what the intention of this was, but it is always TRUE.  Kept for posterity. <JAISON>
m_pAlarmData^.AlarmState := 0;	// Set the initial alarm state to 0, this blinks the alarm logo on the HMI when alarms are active. <JAISON>
END_METHOD

(* ---------------------------------------------------------------------------
Func name   : 	ResetAlarms
Description : 	Resets all state/ack flags in the interface alarm array and
				clears the active alarm counter.
Inputs      :	None
Returns     : 	None
Notes       : 	This routine is intended to clear the alarm interface in the event
				the function block is disabled.
--------------------------------------------------------------------------- *)

METHOD ResetAlarms
VAR_INPUT
END_VAR
VAR
	i		: INT;	// Alarm list index
END_VAR
// Iterate over the interface alarm array and RESET all state/ack flags
FOR i:=0 TO TO_INT(m_numAlarms) - 1 BY 1 DO
 
	// Reset the alarm interface array
	m_pAlarmData^.Alarm[i].state := FALSE;
	m_pAlarmData^.Alarm[i].ack := FALSE;

END_FOR;

// Reset common alarm data to default values <JAISON>
m_pAlarmData^.NumOfActiveAlarms := 0;
m_pAlarmData^.RefreshAlarms := TRUE;
m_pAlarmData^.AlarmState := 0;
END_METHOD

(* ---------------------------------------------------------------------------
Func name   : 	UpdateAlarms
Description : 	Iterates over the interface alarm array and updates the state
				and ack flags to match the internal alarm list.  Maintans an
				active alarm counter which is required by the interface.
Inputs      :	None
Returns     : 	None
Notes       : 	
--------------------------------------------------------------------------- *)

METHOD UpdateAlarms
VAR_INPUT
END_VAR
VAR
	m_pAlarms				: POINTER TO ARRAY[0.._ALARM_ARRAY_MAX_SIZE] OF TAlarmType;	// Alarm Data
	
	i						: INT;		// Alarm List Index
	j						: INT;		// Device Id List Index
	m_notAcked				: BOOL;		// Flag which is TRUE when at least one active alarm is not acked

	m_HighestActivePriority	: UINT;		// Value of the highest priority within a sub group of Device IDs
	m_NumDeviceIdTypes		: INT;		// Number of similar Device IDs used to iterate over each sub group
	
	m_NumActiveInterface 	: UINT;		// Counter of the number of active interface alarms which can now differ
										// from the number of internal alarms IF we are ignoring lower priority
END_VAR
// Assume that no alarms are active and NOT acked
 m_notAcked := FALSE;

// Ensure alarm interface has been initialized
IF (m_numAlarms > 0) THEN

	// Get the system alarms list
	m_pAlarms := m_pAlarmHandler^.GetAlarms();	

	//Ignore all lower priority alarms if filter flag is TRUE
	IF (m_filterPriority) THEN
	
	// reset active alarm counter
	m_NumActiveInterface := 0;

	// Iterate over the interface alarm array and update the state/ack flags
	FOR i:=0 TO TO_INT(m_numAlarms) - 1 BY 1 DO
			
		m_NumDeviceIdTypes := TO_INT(m_pAlarmHandler^.GetNumOfDeviceId(m_pAlarms^[i].code.code.devId));
			
		// Assume highest active alarm priority is the lowest
		m_HighestActivePriority := 0;
				
		// Iterate over all similar Device IDs
		FOR j:=(i + (m_NumDeviceIdTypes - 1)) TO i BY -1 DO
				
			// Set the highest active priority if the alarm is active and higher than the current value
			IF ((m_pAlarms^[j].state = TRUE) AND (f_GetFaultCodePriority(m_pAlarms^[j].code.code.faultCode) > m_HighestActivePriority)) THEN
				m_HighestActivePriority := f_GetFaultCodePriority(m_pAlarms^[j].code.code.faultCode);
			END_IF
				
			// If the current fault code priority is less than the highest active priority
			// for the current Device ID Ignore its state.
			IF (f_GetFaultCodePriority(m_pAlarms^[j].code.code.faultCode) < m_HighestActivePriority) THEN
						
				m_pAlarmData^.Alarm[j].state := FALSE;
					
			// Otherwise copy the alarm state
			ELSE
						
				m_pAlarmData^.Alarm[j].state := m_pAlarms^[j].state;
				
				// incirment the active alarm counter	
				IF (m_pAlarms^[j].state = TRUE) THEN
					m_NumActiveInterface := m_NumActiveInterface + 1;
				END_IF
					
			END_IF
				
		END_FOR
				
		// Skip to the next Device ID
		i := i + (m_NumDeviceIdTypes - 1);
		
		// Flag is there is AT LEAST ONE alarm which is active and not acked
		IF ((m_pAlarmData^.Alarm[i].state) AND (NOT  m_pAlarmData^.Alarm[i].ack)) THEN
			 m_notAcked := TRUE;
		 END_IF	
		// Reset acknowledge if the alarm becomes inactive
		IF ((m_pAlarmData^.Alarm[i].ack) AND (NOT m_pAlarmData^.Alarm[i].state)) THEN
			m_pAlarmData^.Alarm[i].ack := FALSE;
		END_IF
	
	END_FOR;
	
	// Set the number of active alarms
	m_pAlarmData^.NumOfActiveAlarms := TO_INT(m_NumActiveInterface);
	
	//Simply copy all alarm states if filter flag is FALSE
	ELSE

		// Iterate over the interface alarm array and update the state/ack flags
		FOR i:=0 TO TO_INT(m_numAlarms) - 1 BY 1 DO
			
			m_pAlarmData^.Alarm[i].state := m_pAlarms^[i].state;
			
			
			// Flag is there is AT LEAST ONE alarm which is active and not acked
			IF ((m_pAlarmData^.Alarm[i].state) AND (NOT  m_pAlarmData^.Alarm[i].ack)) THEN
			 	m_notAcked := TRUE;
		 	END_IF
			// Reset acknowledge if the alarm becomes inactive
			IF ((m_pAlarmData^.Alarm[i].ack) AND (NOT m_pAlarmData^.Alarm[i].state)) THEN
				m_pAlarmData^.Alarm[i].ack := FALSE;
			END_IF
	
		END_FOR;
	
		// Set the number of active alarms
		m_pAlarmData^.NumOfActiveAlarms := TO_INT(m_pAlarmHandler^.GetNumOfActiveAlarms());
	
	END_IF
	
END_IF

// Update the Alarm state which is used by the HMI to change the icon depending on number of active alarms and their ack status <JAISON>
IF (m_pAlarmData^.NumOfActiveAlarms > 0) THEN
	IF (m_notAcked) THEN
		m_pAlarmData^.AlarmState := 2;	// ACTIVE ALARMS WITH AT LEAST 1 UNACKED - AlarmState = 2
	ELSE
		m_pAlarmData^.AlarmState := 1;	// ACTIVE ALARMS WITH ALL ACKED - AlarmState = 1
	END_IF
ELSE
	m_pAlarmData^.AlarmState := 0;		// NO ACTIVE ALARMS - AlarmState = 0
END_IF
END_METHOD

END_FUNCTION_BLOCK

// 20 Program Organization Units/Command Interface/Interfaces/i_commandHandler
(*AUTHOR:			Jaison Schaab*)
(*DATE:				July. 22 / 2020*)
(*DESCRIPTION: 		This is a standardized interface used by the FSM function
					block to handle generated actions*)
					
(*NOTES:      	 	All methods definied by this interface are required to
					be implimented by the user defined action handler
					function block.  Each methods inputs/outputs need
					to match exactly what is defined by the interface.
					
					The FSM requires the user defined function block which
					impliments this interface  to be passed into its 
					constructor upon instantiation.*)
					
INTERFACE i_commandHandler

(* ---------------------------------------------------------------------------
Func name   : 	CommandDone
Description : 	This method is a standardized handler for each command done
				action generated by the command interface.  This method will
				be called ONCE each time a command is finished.
Inputs      :	pCurrentCommand	-	pointer to the instantiation of the FSM object
Returns     : 	BOOL			- 	result of function (FALSE = Fault)
Notes       : 	The approach of using an interface enables the user 
				of the command interface to define and handle actions 
				based on their design and implementation.
				
				Return FALSE to fault the command interface and trasition
				to the fault state, TRUE to return to the ready state and
				process the next command.
			
				The ONLY commands that need to be processed are the ones defined
				by the used of the class (ie. command ENUM > 0).  The default
				commands of RESET (-1) and NONE (0) do NOT need to be handled here.
				
				If the command interface is Faulted, the Reset method MUST
				be called to clear the buffers and restore command handling.
--------------------------------------------------------------------------- *)

METHOD CommandDone : BOOL
VAR_INPUT
	pCurrentCommand		: POINTER TO TControlCommandBuffer;
END_VAR
END_METHOD

(* ---------------------------------------------------------------------------
Func name   : 	CommandRunning
Description : 	This method is a standardized handler for each command running
				action generated by the command interface.  This method will
				be called each plc scan while a command is running.
Inputs      :	pCurrentCommand	-	pointer to the instantiation of the FSM object
Returns     : 	BOOL			- 	TRUE = DONE, FALSE = CONTINUE PROCESSING
Notes       : 	The approach of using an interface enables the user 
				of the command interface to define and handle actions 
				based on their design and implementation.
				
				Return TRUE to signal the completion of the command and
				run the command done method.  Return FALSE to continue
				running the current command.
				
				If a fault occurs use the "Fault()" method to send the FSM to
				the Fault state.
				
				The ONLY commands that need to be processed are the ones defined
				by the used of the class (ie. command ENUM > 0).  The default
				commands of RESET (-1) and NONE (0) do NOT need to be handled here.
				
				If the command interface is Faulted, the Reset method MUST
				be called to clear the buffers and restore command handling.
--------------------------------------------------------------------------- *)

METHOD CommandRunning : BOOL
VAR_INPUT
	pCurrentCommand		: POINTER TO TControlCommandBuffer;
END_VAR
END_METHOD

(* ---------------------------------------------------------------------------
Func name   : 	CommandStart
Description : 	This method is a standardized handler for each command start
				action generated by the command interface.  This method will
				be called ONCE each time a command is started.
Inputs      :	pCurrentCommand	-	pointer to the instantiation of the FSM object
Returns     : 	BOOL			- 	result of function (FALSE = Fault)
Notes       : 	The approach of using an interface enables the user 
				of the command interface to define and handle actions 
				based on their design and implementation.
				
				Return FALSE to fault the command interface and trasition
				to the fault state, TRUE to return to the ready state and
				process the next command.
				
				The ONLY commands that need to be processed are the ones defined
				by the used of the class (ie. command ENUM > 0).  The default
				commands of RESET (-1) and NONE (0) do NOT need to be handled here.
				
				If the command interface is Faulted, the Reset method MUST
				be called to clear the buffers and restore command handling.
--------------------------------------------------------------------------- *)

METHOD CommandStart : BOOL
VAR_INPUT
	pCurrentCommand		: POINTER TO TControlCommandBuffer;
END_VAR
END_METHOD

(* ---------------------------------------------------------------------------
Func name   : 	Fault
Description : 	This method is a standardized handler for a Fault command
				action generated by the command interface.  This method will
				be called ONCE each time a the interface is faulted.
Inputs      :	None
Returns     : 	None
Notes       : 	The approach of using an interface enables the user 
				of the command interface to define and handle actions 
				based on their design and implementation.
				
				Use this method to perform any required actions on local 
				class member variables needed when the interface is faulted.
--------------------------------------------------------------------------- *)

METHOD Fault
VAR_INPUT
END_VAR
END_METHOD

(* ---------------------------------------------------------------------------
Func name   : 	Reset
Description : 	This method is a standardized handler for a Reset command
				action generated by the command interface.  This method will
				be called ONCE each time a the interface is reset.
Inputs      :	None
Returns     : 	None
Notes       : 	The approach of using an interface enables the user 
				of the command interface to define and handle actions 
				based on their design and implementation.
				
				Use this method to reset any local class member variables
				or objects that need to be reset outside of the standard
				command interface class.
				
				A reset command will have already cleared the command buffers
				and control FSM before this method is executed.
--------------------------------------------------------------------------- *)

METHOD Reset
VAR_INPUT
END_VAR
END_METHOD

END_INTERFACE

// 20 Program Organization Units/Command Interface/fb_CommandInterface
(*AUTHOR:			Jaison Schaab*)
(*DATE:				July 28 / 2020*)
(*DESCRIPTION: 		This Function Block provides the standard base functionality for
					a command/response control interface including a FIFO buffer
					and state machine to handle buffered commands.*)
					
(*NOTES:			The user of the command interface function block is required to define the following:

					COMMAND ENUM of TYPE TControlCommand (INT) 								- 	List of defined commands starting at 1
																								User must define the default commands of RESET (-1) and NONE (0)
					COMMAND PARM UNION of TYPE TControlCommandParms (ARRAY[1..10] OF WORD) 	- 	Union which overlays the required command parms over the standard
																								raw parm array of 10 WORDS (TControlCommandParms)
					RESPONSE ENUM of TYPE TControlResponse (INT) 							- 	List of defined command resonses starting at 1
																								User must define the default responses of FAULT (-2), BUSY (-1) and READY (0)
					
					A valid user defined command is INT greater than 0, starting at 1.  The RESET (-1) command is automatically handled by the
					interface and will clear the FIFO buffer, reset the FSM and call the user defined Reset() interface function.
																								
					****WAGO does NOT allow the ENUMERATION types to be defined as a non-registered type (ex. TControlCommand)
						To work around this simply define the required ENUMERATIONS as INT and remove the 
						"{attribute 'strict'}" from the header so that the system will correlate the non-registered types****
					
					CommandStart function block  			- 	user defined function block required by the i_commandHandler interface and
																will be called ONCE each time a command is started.
																
					CommandRunning function block  			- 	user defined function block required by the i_commandHandler interface and
																will be called each plc scan while a command is running.
																
					CommandDone function block  			- 	user defined function block required by the i_commandHandler interface and
																will be called ONCE each time a command is finished.
																
					Reset function block  					- 	user defined function block required by the i_commandHandler interface and
																will be called ONCE each time a the interface is reset.
																							
					
					****TO SEND COMMANDS to the interface use the "SendCommand" method.****
					
					****Ensure that the "CMD_Init" method is run in the constructor or the class using the command interface:
					
						// Initialize the command interface
						Init(commandHandler:= THIS^);
						
						Ensure that the "UpdateCommandInterface" method is cyclically called by the class using the command interface.****
*)

(*UPDATE: 		April 20 2021 - Jaison Schaab

				Integrated the Beckhoff FB_MemRingBuffer in place of the Wago FIFO buffer and made the code changes accordingly.  The 
				buffer is now defined as an array of BYTEs instead of and array of TControlCommandBuffer because beckhoff pads each
				data set is complemented with additional information (4BYTES), so that it can be located later; This means that
				the BYTE size of the buffer is now computed in the constants based on a new entry which defines the M_COMMAND_BUFFER_NUM_ENTRIES.
				
				I have modifed the check in CMD_SendCommand to use the num entries rather than buffer size as this is easier to understand
				and accomplishes the same functionality in not allowing more entires than buffer size.  I tested the buffer to max size and
				confirmed no errors are present when trying to overflow the buffer with the new logic.

				Code Is fully tested and functional.	
*)

(*UPDATE: 		March 03 2021 - Graham Hunter

				Ported over fb_CommandInterface code from ECP to TwinCAT. Had to use MEMSET and MEMCPY from TwinCAT for the equivalent functions in Wago.
				NEED TO TEST WITH THE TWINCAT FB_MemRingBufferEx. See FB_MemRingBufferEx sample code in Beckhoff InfoSys!
*)

FUNCTION_BLOCK fb_CommandInterface IMPLEMENTS i_actionHandler
VAR_INPUT
	xEnable							: BOOL;
END_VAR
VAR_OUTPUT
	xBusy							: BOOL;								// TRUE = Command is executing, FALSE = No command running
	xDone							: BOOL;								// TRUE = Command is done, FALSE = Command is running 
	xFault							: BOOL;								// TRUE = FSM faulted (must reset), FALSE = No fault present
END_VAR
VAR
	// Internal Command Variables
	m_ControlEnabled				: BOOL;								// Flag to enable control logic
	m_CurrentCommand				: TControlCommandBuffer;			// Current commmand being removed from the FIFO buffer
	
	m_pCmdTraceTable				: POINTER TO TControlCommandBuffer;	// Pointer to the trace table
	m_CmdTraceTableSize				: UINT;								// Size of the trace table array in BYTES
	
	// Event Triggers

	m_EnableTrigger					: R_TRIG;							// Control enable event trigger
	m_DisableTrigger				: F_TRIG;							// Control disable event trigger
	m_CommandDoneTrigger			: R_TRIG;							// Command done event trigger
	
